  MoveL 10746 to (-26.41, 164.46, 144.49) mm, rotated rx 180 ry 0 rz 180 deg; joints [-138.58, 73.769, -86.473, 137.874, 80.508, 8.483]
  MoveL 10747 to (-26.41, 164.46, 144.49) mm, rotated rx 180 ry 0 rz 180 deg; joints [-138.58, 73.769, -86.473, 137.874, 80.508, 8.483]
  Call Extruder(786.45061)
  MoveL 10748 to (-26.72, 164.41, 144.49) mm, rotated rx 180 ry 0 rz 180 deg; joints [-138.635, 73.783, -86.46, 137.932, 80.52, 8.455]
  MoveL 10749 to (-26.72, 164.41, 144.49) mm, rotated rx 180 ry 0 rz 180 deg; joints [-138.635, 73.783, -86.46, 137.932, 80.52, 8.455]
  Call Extruder(786.61308)
  MoveL 10750 to (-27.03, 164.37, 144.49) mm, rotated rx -180 ry 0 rz -180 deg; joints [-138.69, 73.796, -86.447, 137.99, 80.531, 8.428]
  MoveL 10751 to (-27.03, 164.37, 144.49) mm, rotated rx -180 ry 0 rz -180 deg; joints [-138.69, 73.796, -86.447, 137.99, 80.531, 8.428]
  Call Extruder(786.74701)
  MoveL 10752 to (-27.27, 164.32, 144.49) mm, rotated rx -180 ry 0 rz 180 deg; joints [-138.736, 73.807, -86.437, 138.039, 80.54, 8.407]
  MoveL 10753 to (-27.27, 164.32, 144.49) mm, rotated rx -180 ry 0 rz 180 deg; joints [-138.736, 73.807, -86.437, 138.039, 80.54, 8.407]
  Call Extruder(786.88155)
  MoveL 10754 to (-27.52, 164.27, 144.49) mm, rotated rx -180 ry 0 rz 180 deg; joints [-138.783, 73.817, -86.426, 138.088, 80.549, 8.385]
  MoveL 10755 to (-27.52, 164.27, 144.49) mm, rotated rx -180 ry 0 rz 180 deg; joints [-138.783, 73.817, -86.426, 138.088, 80.549, 8.385]
  Call Extruder(787.01669)
  MoveL 10756 to (-27.77, 164.22, 144.49) mm, rotated rx 180 ry 0 rz -180 deg; joints [-138.829, 73.828, -86.416, 138.137, 80.557, 8.363]
  MoveL 10757 to (-27.77, 164.22, 144.49) mm, rotated rx 180 ry 0 rz -180 deg; joints [-138.829, 73.828, -86.416, 138.137, 80.557, 8.363]
  Call Extruder(787.15245)
  MoveL 10758 to (-28.02, 164.17, 144.49) mm, rotated rx -180 ry 0 rz 180 deg; joints [-138.875, 73.838, -86.406, 138.185, 80.566, 8.342]
  MoveL 10759 to (-28.02, 164.17, 144.49) mm, rotated rx -180 ry 0 rz 180 deg; joints [-138.875, 73.838, -86.406, 138.185, 80.566, 8.342]
  Call Extruder(787.28882)
  MoveL 10760 to (-28.27, 164.12, 144.49) mm, rotated rx -180 ry 0 rz 180 deg; joints [-138.921, 73.848, -86.395, 138.234, 80.575, 8.32]
  MoveL 10761 to (-28.27, 164.12, 144.49) mm, rotated rx -180 ry 0 rz 180 deg; joints [-138.921, 73.848, -86.395, 138.234, 80.575, 8.32]
  Call Extruder(787.42580)
  MoveL 10762 to (-28.52, 164.07, 144.49) mm, rotated rx -180 ry 0 rz 180 deg; joints [-138.967, 73.859, -86.385, 138.283, 80.584, 8.298]
  MoveL 10763 to (-28.52, 164.07, 144.49) mm, rotated rx -180 ry 0 rz 180 deg; joints [-138.967, 73.859, -86.385, 138.283, 80.584, 8.298]
  Call Extruder(787.56338)
  MoveL 10764 to (-28.77, 164.02, 144.49) mm, rotated rx -180 ry 0 rz 180 deg; joints [-139.013, 73.869, -86.375, 138.331, 80.593, 8.277]
  MoveL 10765 to (-28.77, 164.02, 144.49) mm, rotated rx -180 ry 0 rz 180 deg; joints [-139.013, 73.869, -86.375, 138.331, 80.593, 8.277]
  Call Extruder(787.67710)
  MoveL 10766 to (-28.97, 163.97, 144.49) mm, rotated rx -180 ry 0 rz -180 deg; joints [-139.052, 73.878, -86.366, 138.371, 80.6, 8.259]
  MoveL 10767 to (-28.97, 163.97, 144.49) mm, rotated rx -180 ry 0 rz -180 deg; joints [-139.052, 73.878, -86.366, 138.371, 80.6, 8.259]
  Call Extruder(787.79127)
  MoveL 10768 to (-29.18, 163.93, 144.49) mm, rotated rx -180 ry 0 rz 180 deg; joints [-139.09, 73.886, -86.358, 138.412, 80.607, 8.241]
  MoveL 10769 to (-29.18, 163.93, 144.49) mm, rotated rx -180 ry 0 rz 180 deg; joints [-139.09, 73.886, -86.358, 138.412, 80.607, 8.241]
  Call Extruder(787.90589)
  MoveL 10770 to (-29.38, 163.88, 144.49) mm, rotated rx 180 ry 0 rz 180 deg; joints [-139.128, 73.895, -86.349, 138.452, 80.614, 8.224]
  MoveL 10771 to (-29.38, 163.88, 144.49) mm, rotated rx 180 ry 0 rz 180 deg; joints [-139.128, 73.895, -86.349, 138.452, 80.614, 8.224]
  Call Extruder(788.02096)
  MoveL 10772 to (-29.59, 163.84, 144.49) mm, rotated rx 180 ry 0 rz 180 deg; joints [-139.166, 73.903, -86.341, 138.492, 80.621, 8.206]
  MoveL 10773 to (-29.59, 163.84, 144.49) mm, rotated rx 180 ry 0 rz 180 deg; joints [-139.166, 73.903, -86.341, 138.492, 80.621, 8.206]
  Call Extruder(788.14320)
  MoveL 10774 to (-29.8, 163.78, 144.49) mm, rotated rx -180 ry 0 rz -180 deg; joints [-139.208, 73.911, -86.332, 138.536, 80.628, 8.188]
  MoveL 10775 to (-29.8, 163.78, 144.49) mm, rotated rx -180 ry 0 rz -180 deg; joints [-139.208, 73.911, -86.332, 138.536, 80.628, 8.188]
  Call Extruder(788.27288)
  MoveL 10776 to (-30.02, 163.72, 144.49) mm, rotated rx -180 ry 0 rz 180 deg; joints [-139.253, 73.92, -86.324, 138.583, 80.634, 8.17]
  MoveL 10777 to (-30.02, 163.72, 144.49) mm, rotated rx -180 ry 0 rz 180 deg; joints [-139.253, 73.92, -86.324, 138.583, 80.634, 8.17]
  Call Extruder(788.40312)
  MoveL 10778 to (-30.25, 163.65, 144.49) mm, rotated rx -180 ry 0 rz 180 deg; joints [-139.298, 73.928, -86.316, 138.63, 80.64, 8.151]
  MoveL 10779 to (-30.25, 163.65, 144.49) mm, rotated rx -180 ry 0 rz 180 deg; joints [-139.298, 73.928, -86.316, 138.63, 80.64, 8.151]
  Call Extruder(788.53393)
  MoveL 10780 to (-30.47, 163.58, 144.49) mm, rotated rx -180 ry 0 rz 180 deg; joints [-139.343, 73.937, -86.307, 138.677, 80.647, 8.132]
  MoveL 10781 to (-30.47, 163.58, 144.49) mm, rotated rx -180 ry 0 rz 180 deg; joints [-139.343, 73.937, -86.307, 138.677, 80.647, 8.132]
  Call Extruder(788.66530)
  MoveL 10782 to (-30.69, 163.51, 144.49) mm, rotated rx -180 ry 0 rz 180 deg; joints [-139.388, 73.945, -86.299, 138.724, 80.653, 8.114]
  MoveL 10783 to (-30.69, 163.51, 144.49) mm, rotated rx -180 ry 0 rz 180 deg; joints [-139.388, 73.945, -86.299, 138.724, 80.653, 8.114]
  Call Extruder(788.77719)
  MoveL 10784 to (-30.88, 163.45, 144.49) mm, rotated rx -180 ry 0 rz 180 deg; joints [-139.427, 73.952, -86.292, 138.764, 80.658, 8.098]
  MoveL 10785 to (-30.88, 163.45, 144.49) mm, rotated rx -180 ry 0 rz 180 deg; joints [-139.427, 73.952, -86.292, 138.764, 80.658, 8.098]
  Call Extruder(788.88953)
  MoveL 10786 to (-31.07, 163.39, 144.49) mm, rotated rx -180 ry 0 rz 180 deg; joints [-139.465, 73.959, -86.285, 138.804, 80.663, 8.083]
  MoveL 10787 to (-31.07, 163.39, 144.49) mm, rotated rx -180 ry 0 rz 180 deg; joints [-139.465, 73.959, -86.285, 138.804, 80.663, 8.083]
  Call Extruder(789.00231)
  MoveL 10788 to (-31.26, 163.33, 144.49) mm, rotated rx 180 ry 0 rz -180 deg; joints [-139.504, 73.966, -86.278, 138.844, 80.668, 8.067]
  MoveL 10789 to (-31.26, 163.33, 144.49) mm, rotated rx 180 ry 0 rz -180 deg; joints [-139.504, 73.966, -86.278, 138.844, 80.668, 8.067]
  Call Extruder(789.11553)
  MoveL 10790 to (-31.45, 163.27, 144.49) mm, rotated rx 180 ry 0 rz -180 deg; joints [-139.542, 73.973, -86.271, 138.885, 80.673, 8.052]
  MoveL 10791 to (-31.45, 163.27, 144.49) mm, rotated rx 180 ry 0 rz -180 deg; joints [-139.542, 73.973, -86.271, 138.885, 80.673, 8.052]
  Call Extruder(789.22920)
  MoveL 10792 to (-31.64, 163.21, 144.49) mm, rotated rx 180 ry 0 rz 180 deg; joints [-139.581, 73.979, -86.264, 138.925, 80.678, 8.036]
  MoveL 10793 to (-31.64, 163.21, 144.49) mm, rotated rx 180 ry 0 rz 180 deg; joints [-139.581, 73.979, -86.264, 138.925, 80.678, 8.036]
  Call Extruder(789.41118)
  MoveL 10794 to (-31.93, 163.09, 144.49) mm, rotated rx -180 ry 0 rz -180 deg; joints [-139.645, 73.989, -86.254, 138.991, 80.684, 8.013]
  MoveL 10795 to (-31.93, 163.09, 144.49) mm, rotated rx -180 ry 0 rz -180 deg; joints [-139.645, 73.989, -86.254, 138.991, 80.684, 8.013]
  Call Extruder(789.59392)
  MoveL 10796 to (-32.22, 162.96, 144.49) mm, rotated rx -180 ry 0 rz 180 deg; joints [-139.709, 73.999, -86.244, 139.057, 80.69, 7.989]
  MoveL 10797 to (-32.22, 162.96, 144.49) mm, rotated rx -180 ry 0 rz 180 deg; joints [-139.709, 73.999, -86.244, 139.057, 80.69, 7.989]
  Call Extruder(789.76433)
  MoveL 10798 to (-32.49, 162.85, 144.49) mm, rotated rx 180 ry 0 rz -180 deg; joints [-139.768, 74.007, -86.235, 139.119, 80.695, 7.968]
  MoveL 10799 to (-32.49, 162.85, 144.49) mm, rotated rx 180 ry 0 rz -180 deg; joints [-139.768, 74.007, -86.235, 139.119, 80.695, 7.968]
  Call Extruder(789.92231)
  MoveL 10800 to (-32.74, 162.74, 144.49) mm, rotated rx 180 ry 0 rz 180 deg; joints [-139.823, 74.016, -86.227, 139.176, 80.699, 7.948]
  MoveL 10801 to (-32.74, 162.74, 144.49) mm, rotated rx 180 ry 0 rz 180 deg; joints [-139.823, 74.016, -86.227, 139.176, 80.699, 7.948]
  Call Extruder(790.08088)
  MoveL 10802 to (-32.99, 162.64, 144.49) mm, rotated rx -180 ry 0 rz -180 deg; joints [-139.878, 74.024, -86.219, 139.233, 80.704, 7.929]
  MoveL 10803 to (-32.99, 162.64, 144.49) mm, rotated rx -180 ry 0 rz -180 deg; joints [-139.878, 74.024, -86.219, 139.233, 80.704, 7.929]
  Call Extruder(790.28705)
  MoveL 10804 to (-33.29, 162.46, 144.49) mm, rotated rx 180 ry 0 rz 180 deg; joints [-139.953, 74.032, -86.211, 139.31, 80.706, 7.906]
  MoveL 10805 to (-33.29, 162.46, 144.49) mm, rotated rx 180 ry 0 rz 180 deg; joints [-139.953, 74.032, -86.211, 139.31, 80.706, 7.906]
  Call Extruder(790.49399)
  MoveL 10806 to (-33.6, 162.29, 144.49) mm, rotated rx -180 ry 0 rz -180 deg; joints [-140.028, 74.04, -86.202, 139.387, 80.708, 7.883]
  MoveL 10807 to (-33.6, 162.29, 144.49) mm, rotated rx -180 ry 0 rz -180 deg; joints [-140.028, 74.04, -86.202, 139.387, 80.708, 7.883]
  Call Extruder(790.70172)
  MoveL 10808 to (-33.9, 162.11, 144.49) mm, rotated rx 180 ry 0 rz 180 deg; joints [-140.103, 74.048, -86.194, 139.463, 80.71, 7.86]
  MoveL 10809 to (-33.9, 162.11, 144.49) mm, rotated rx 180 ry 0 rz 180 deg; joints [-140.103, 74.048, -86.194, 139.463, 80.71, 7.86]
  Call Extruder(790.91022)
  MoveL 10810 to (-34.21, 161.94, 144.49) mm, rotated rx 180 ry 0 rz 180 deg; joints [-140.178, 74.056, -86.186, 139.54, 80.712, 7.837]
  MoveL 10811 to (-34.21, 161.94, 144.49) mm, rotated rx 180 ry 0 rz 180 deg; joints [-140.178, 74.056, -86.186, 139.54, 80.712, 7.837]
  Call Extruder(791.08976)
  MoveL 10812 to (-34.45, 161.76, 144.49) mm, rotated rx 180 ry 0 rz 180 deg; joints [-140.244, 74.061, -86.181, 139.607, 80.711, 7.82]
  MoveL 10813 to (-34.45, 161.76, 144.49) mm, rotated rx 180 ry 0 rz 180 deg; joints [-140.244, 74.061, -86.181, 139.607, 80.711, 7.82]
  Call Extruder(791.42319)
  MoveL 10814 to (-34.9, 161.43, 144.49) mm, rotated rx -180 ry 0 rz -180 deg; joints [-140.366, 74.07, -86.171, 139.732, 80.708, 7.788]
  MoveL 10815 to (-34.9, 161.43, 144.49) mm, rotated rx -180 ry 0 rz -180 deg; joints [-140.366, 74.07, -86.171, 139.732, 80.708, 7.788]
  Call Extruder(791.75781)
  MoveL 10816 to (-35.35, 161.1, 144.49) mm, rotated rx 180 ry 0 rz 180 deg; joints [-140.489, 74.079, -86.162, 139.857, 80.706, 7.756]
  Call Extruder(792.58572)
  MoveL 10817 to (-36.39, 160.19, 144.49) mm, rotated rx -180 ry 0 rz -180 deg; joints [-140.797, 74.094, -86.147, 140.17, 80.688, 7.686]
  Call Extruder(793.10708)
  MoveL 10818 to (-36.97, 159.54, 144.49) mm, rotated rx 180 ry 0 rz -180 deg; joints [-140.993, 74.096, -86.144, 140.368, 80.665, 7.651]
  Set speed (130.0 mm/s)
  MoveL 10819 to (-38.97, 156.79, 144.49) mm, rotated rx 180 ry 0 rz 180 deg; joints [-141.763, 74.086, -86.155, 141.139, 80.548, 7.538]
  MoveL 10820 to (-38.97, 156.78, 153.89) mm, rotated rx -180 ry 0 rz 180 deg; joints [-141.763, 75.445, -87.86, 141.102, 80.278, 7.758]
  Call Extruder(791.10708)
  Set speed (40.0 mm/s)
  MoveL 10821 to (-38.97, 156.78, 153.89) mm, rotated rx -180 ry 0 rz 180 deg; joints [-141.763, 75.445, -87.86, 141.102, 80.278, 7.758]
  Call Extruder(0.00000)
  Set speed (130.0 mm/s)
  MoveL 10822 to (-31.64, 163.21, 153.89) mm, rotated rx 180 ry 0 rz -180 deg; joints [-139.581, 75.337, -87.97, 138.886, 80.415, 8.268]
  Call Extruder(2.00000)
  Set speed (40.0 mm/s)
  MoveL 10823 to (-31.64, 163.21, 153.89) mm, rotated rx 180 ry 0 rz -180 deg; joints [-139.581, 75.337, -87.97, 138.886, 80.415, 8.268]
  Set speed (30.0 mm/s)
  MoveL 10824 to (-31.64, 163.21, 153.89) mm, rotated rx 180 ry 0 rz -180 deg; joints [-139.581, 75.337, -87.97, 138.886, 80.415, 8.268]
  Call Extruder(2.18198)
  MoveL 10825 to (-31.93, 163.09, 153.89) mm, rotated rx -180 ry 0 rz -180 deg; joints [-139.645, 75.347, -87.96, 138.953, 80.421, 8.245]
  MoveL 10826 to (-31.93, 163.09, 153.89) mm, rotated rx -180 ry 0 rz -180 deg; joints [-139.645, 75.347, -87.96, 138.953, 80.421, 8.245]
  Call Extruder(2.36471)
  MoveL 10827 to (-32.22, 162.96, 153.89) mm, rotated rx -180 ry 0 rz -180 deg; joints [-139.709, 75.356, -87.95, 139.019, 80.427, 8.221]
  MoveL 10828 to (-32.22, 162.96, 153.89) mm, rotated rx -180 ry 0 rz -180 deg; joints [-139.709, 75.356, -87.95, 139.019, 80.427, 8.221]
  Call Extruder(2.53265)
  MoveL 10829 to (-32.49, 162.85, 153.89) mm, rotated rx 180 ry 0 rz 180 deg; joints [-139.767, 75.365, -87.941, 139.08, 80.432, 8.199]
  MoveL 10830 to (-32.49, 162.85, 153.89) mm, rotated rx 180 ry 0 rz 180 deg; joints [-139.767, 75.365, -87.941, 139.08, 80.432, 8.199]
  Call Extruder(2.68564)
  MoveL 10831 to (-32.73, 162.75, 153.89) mm, rotated rx -180 ry 0 rz 180 deg; joints [-139.821, 75.373, -87.933, 139.135, 80.436, 8.18]
  MoveL 10832 to (-32.73, 162.75, 153.89) mm, rotated rx -180 ry 0 rz 180 deg; joints [-139.821, 75.373, -87.933, 139.135, 80.436, 8.18]
  Call Extruder(2.83919)
  MoveL 10833 to (-32.97, 162.65, 153.89) mm, rotated rx 180 ry 0 rz 180 deg; joints [-139.874, 75.381, -87.925, 139.19, 80.441, 8.16]
  MoveL 10834 to (-32.97, 162.65, 153.89) mm, rotated rx 180 ry 0 rz 180 deg; joints [-139.874, 75.381, -87.925, 139.19, 80.441, 8.16]
  Call Extruder(3.04828)
  MoveL 10835 to (-33.28, 162.47, 153.89) mm, rotated rx -180 ry 0 rz 180 deg; joints [-139.95, 75.389, -87.917, 139.269, 80.442, 8.137]
  MoveL 10836 to (-33.28, 162.47, 153.89) mm, rotated rx -180 ry 0 rz 180 deg; joints [-139.95, 75.389, -87.917, 139.269, 80.442, 8.137]
  Call Extruder(3.25817)
  MoveL 10837 to (-33.59, 162.29, 153.89) mm, rotated rx -180 ry 0 rz -180 deg; joints [-140.026, 75.398, -87.909, 139.347, 80.444, 8.113]
  MoveL 10838 to (-33.59, 162.29, 153.89) mm, rotated rx -180 ry 0 rz -180 deg; joints [-140.026, 75.398, -87.909, 139.347, 80.444, 8.113]
  Call Extruder(3.46884)
  MoveL 10839 to (-33.89, 162.11, 153.89) mm, rotated rx -180 ry 0 rz -180 deg; joints [-140.102, 75.406, -87.9, 139.425, 80.446, 8.09]
  MoveL 10840 to (-33.89, 162.11, 153.89) mm, rotated rx -180 ry 0 rz -180 deg; joints [-140.102, 75.406, -87.9, 139.425, 80.446, 8.09]
  Call Extruder(3.68030)
  MoveL 10841 to (-34.2, 161.93, 153.89) mm, rotated rx -180 ry 0 rz 180 deg; joints [-140.178, 75.414, -87.892, 139.503, 80.448, 8.066]
  MoveL 10842 to (-34.2, 161.93, 153.89) mm, rotated rx -180 ry 0 rz 180 deg; joints [-140.178, 75.414, -87.892, 139.503, 80.448, 8.066]
  Call Extruder(3.88506)
  MoveL 10843 to (-34.48, 161.73, 153.89) mm, rotated rx -180 ry 0 rz -180 deg; joints [-140.253, 75.42, -87.886, 139.579, 80.447, 8.045]
  MoveL 10844 to (-34.48, 161.73, 153.89) mm, rotated rx -180 ry 0 rz -180 deg; joints [-140.253, 75.42, -87.886, 139.579, 80.447, 8.045]
  Call Extruder(4.20602)
  MoveL 10845 to (-34.92, 161.42, 153.89) mm, rotated rx 180 ry 0 rz 180 deg; joints [-140.371, 75.429, -87.877, 139.7, 80.444, 8.014]
  MoveL 10846 to (-34.92, 161.42, 153.89) mm, rotated rx 180 ry 0 rz 180 deg; joints [-140.371, 75.429, -87.877, 139.7, 80.444, 8.014]
  Call Extruder(4.52807)
  MoveL 10847 to (-35.35, 161.1, 153.89) mm, rotated rx 180 ry 0 rz 180 deg; joints [-140.489, 75.438, -87.867, 139.82, 80.442, 7.982]
  Call Extruder(5.35599)
  MoveL 10848 to (-36.39, 160.19, 153.89) mm, rotated rx -180 ry 0 rz 180 deg; joints [-140.797, 75.453, -87.852, 140.133, 80.422, 7.911]
  Call Extruder(6.18392)
  MoveL 10849 to (-37.3, 159.15, 153.89) mm, rotated rx 180 ry 0 rz 180 deg; joints [-141.109, 75.457, -87.848, 140.447, 80.385, 7.854]
  Call Extruder(6.34862)
  MoveL 10850 to (-37.47, 158.93, 153.89) mm, rotated rx -180 ry 0 rz -180 deg; joints [-141.171, 75.456, -87.849, 140.509, 80.375, 7.845]
  MoveL 10851 to (-37.47, 158.93, 153.89) mm, rotated rx -180 ry 0 rz -180 deg; joints [-141.171, 75.456, -87.849, 140.509, 80.375, 7.845]
  Call Extruder(6.67688)
  MoveL 10852 to (-37.79, 158.49, 153.89) mm, rotated rx -180 ry 0 rz 180 deg; joints [-141.295, 75.454, -87.851, 140.634, 80.356, 7.826]
  MoveL 10853 to (-37.79, 158.49, 153.89) mm, rotated rx -180 ry 0 rz 180 deg; joints [-141.295, 75.454, -87.851, 140.634, 80.356, 7.826]
  Call Extruder(7.00398)
  MoveL 10854 to (-38.11, 158.04, 153.89) mm, rotated rx -180 ry 0 rz -180 deg; joints [-141.419, 75.452, -87.853, 140.758, 80.336, 7.807]
  MoveL 10855 to (-38.11, 158.04, 153.89) mm, rotated rx -180 ry 0 rz -180 deg; joints [-141.419, 75.452, -87.853, 140.758, 80.336, 7.807]
  Call Extruder(7.13851)
  MoveL 10856 to (-38.23, 157.85, 153.89) mm, rotated rx 180 ry 0 rz 180 deg; joints [-141.47, 75.45, -87.855, 140.808, 80.326, 7.802]
  MoveL 10857 to (-38.23, 157.85, 153.89) mm, rotated rx 180 ry 0 rz 180 deg; joints [-141.47, 75.45, -87.855, 140.808, 80.326, 7.802]
  Call Extruder(7.35382)
  MoveL 10858 to (-38.41, 157.53, 153.89) mm, rotated rx -180 ry 0 rz 180 deg; joints [-141.551, 75.447, -87.859, 140.889, 80.309, 7.793]
  MoveL 10859 to (-38.41, 157.53, 153.89) mm, rotated rx -180 ry 0 rz 180 deg; joints [-141.551, 75.447, -87.859, 140.889, 80.309, 7.793]
  Call Extruder(7.56829)
  MoveL 10860 to (-38.59, 157.22, 153.89) mm, rotated rx -180 ry 0 rz -180 deg; joints [-141.632, 75.443, -87.863, 140.97, 80.292, 7.784]
  MoveL 10861 to (-38.59, 157.22, 153.89) mm, rotated rx -180 ry 0 rz -180 deg; joints [-141.632, 75.443, -87.863, 140.97, 80.292, 7.784]
  Call Extruder(7.78192)
  MoveL 10862 to (-38.77, 156.9, 153.89) mm, rotated rx -180 ry 0 rz 180 deg; joints [-141.714, 75.439, -87.866, 141.051, 80.275, 7.775]
  MoveL 10863 to (-38.77, 156.9, 153.89) mm, rotated rx -180 ry 0 rz 180 deg; joints [-141.714, 75.439, -87.866, 141.051, 80.275, 7.775]
  Call Extruder(7.96114)
  MoveL 10864 to (-38.91, 156.63, 153.89) mm, rotated rx -180 ry 0 rz 180 deg; joints [-141.782, 75.435, -87.87, 141.119, 80.26, 7.768]
  MoveL 10865 to (-38.91, 156.63, 153.89) mm, rotated rx -180 ry 0 rz 180 deg; joints [-141.782, 75.435, -87.87, 141.119, 80.26, 7.768]
  Call Extruder(8.10685)
  MoveL 10866 to (-39.01, 156.4, 153.89) mm, rotated rx -180 ry 0 rz -180 deg; joints [-141.837, 75.431, -87.875, 141.173, 80.246, 7.764]
  MoveL 10867 to (-39.01, 156.4, 153.89) mm, rotated rx -180 ry 0 rz -180 deg; joints [-141.837, 75.431, -87.875, 141.173, 80.246, 7.764]
  Call Extruder(8.25205)
  MoveL 10868 to (-39.11, 156.17, 153.89) mm, rotated rx 180 ry 0 rz 180 deg; joints [-141.891, 75.427, -87.879, 141.227, 80.232, 7.761]
  MoveL 10869 to (-39.11, 156.17, 153.89) mm, rotated rx 180 ry 0 rz 180 deg; joints [-141.891, 75.427, -87.879, 141.227, 80.232, 7.761]
  Call Extruder(8.43477)
  MoveL 10870 to (-39.23, 155.88, 153.89) mm, rotated rx 180 ry 0 rz -180 deg; joints [-141.96, 75.421, -87.885, 141.295, 80.213, 7.756]
  MoveL 10871 to (-39.23, 155.88, 153.89) mm, rotated rx 180 ry 0 rz -180 deg; joints [-141.96, 75.421, -87.885, 141.295, 80.213, 7.756]
  Call Extruder(8.61673)
  MoveL 10872 to (-39.35, 155.58, 153.89) mm, rotated rx -180 ry 0 rz 180 deg; joints [-142.029, 75.415, -87.891, 141.363, 80.195, 7.752]
  MoveL 10873 to (-39.35, 155.58, 153.89) mm, rotated rx -180 ry 0 rz 180 deg; joints [-142.029, 75.415, -87.891, 141.363, 80.195, 7.752]
  Call Extruder(8.76407)
  MoveL 10874 to (-39.44, 155.34, 153.89) mm, rotated rx -180 ry 0 rz 180 deg; joints [-142.085, 75.41, -87.896, 141.418, 80.179, 7.749]
  MoveL 10875 to (-39.44, 155.34, 153.89) mm, rotated rx -180 ry 0 rz 180 deg; joints [-142.085, 75.41, -87.896, 141.418, 80.179, 7.749]
  Call Extruder(8.87730)
  MoveL 10876 to (-39.5, 155.15, 153.89) mm, rotated rx -180 ry 0 rz -180 deg; joints [-142.127, 75.405, -87.901, 141.46, 80.166, 7.747]
  MoveL 10877 to (-39.5, 155.15, 153.89) mm, rotated rx -180 ry 0 rz -180 deg; joints [-142.127, 75.405, -87.901, 141.46, 80.166, 7.747]
  Call Extruder(8.99009)
  MoveL 10878 to (-39.56, 154.97, 153.89) mm, rotated rx -180 ry 0 rz -180 deg; joints [-142.169, 75.401, -87.905, 141.501, 80.154, 7.746]
  MoveL 10879 to (-39.56, 154.97, 153.89) mm, rotated rx -180 ry 0 rz -180 deg; joints [-142.169, 75.401, -87.905, 141.501, 80.154, 7.746]
  Call Extruder(9.10244)
  MoveL 10880 to (-39.62, 154.78, 153.89) mm, rotated rx 180 ry 0 rz -180 deg; joints [-142.212, 75.396, -87.91, 141.543, 80.141, 7.744]
  MoveL 10881 to (-39.62, 154.78, 153.89) mm, rotated rx 180 ry 0 rz -180 deg; joints [-142.212, 75.396, -87.91, 141.543, 80.141, 7.744]
  Call Extruder(9.21434)
  MoveL 10882 to (-39.68, 154.59, 153.89) mm, rotated rx 180 ry 0 rz -180 deg; joints [-142.254, 75.392, -87.914, 141.584, 80.128, 7.743]
  MoveL 10883 to (-39.68, 154.59, 153.89) mm, rotated rx 180 ry 0 rz -180 deg; joints [-142.254, 75.392, -87.914, 141.584, 80.128, 7.743]
  Call Extruder(9.33574)
  MoveL 10884 to (-39.75, 154.38, 153.89) mm, rotated rx -180 ry 0 rz 180 deg; joints [-142.3, 75.387, -87.919, 141.629, 80.114, 7.741]
  MoveL 10885 to (-39.75, 154.38, 153.89) mm, rotated rx -180 ry 0 rz 180 deg; joints [-142.3, 75.387, -87.919, 141.629, 80.114, 7.741]
  Call Extruder(9.46653)
  MoveL 10886 to (-39.81, 154.16, 153.89) mm, rotated rx -180 ry 0 rz 180 deg; joints [-142.35, 75.381, -87.925, 141.678, 80.098, 7.74]
  MoveL 10887 to (-39.81, 154.16, 153.89) mm, rotated rx -180 ry 0 rz 180 deg; joints [-142.35, 75.381, -87.925, 141.678, 80.098, 7.74]
  Call Extruder(9.59676)
  MoveL 10888 to (-39.88, 153.94, 153.89) mm, rotated rx -180 ry 0 rz -180 deg; joints [-142.399, 75.376, -87.931, 141.726, 80.083, 7.738]
  MoveL 10889 to (-39.88, 153.94, 153.89) mm, rotated rx -180 ry 0 rz -180 deg; joints [-142.399, 75.376, -87.931, 141.726, 80.083, 7.738]
  Call Extruder(9.72643)
  MoveL 10890 to (-39.95, 153.71, 153.89) mm, rotated rx -180 ry 0 rz 180 deg; joints [-142.449, 75.37, -87.936, 141.775, 80.067, 7.737]
  MoveL 10891 to (-39.95, 153.71, 153.89) mm, rotated rx -180 ry 0 rz 180 deg; joints [-142.449, 75.37, -87.936, 141.775, 80.067, 7.737]
  Call Extruder(9.85553)
  MoveL 10892 to (-40.02, 153.49, 153.89) mm, rotated rx -180 ry 0 rz -180 deg; joints [-142.498, 75.364, -87.942, 141.824, 80.052, 7.735]
  MoveL 10893 to (-40.02, 153.49, 153.89) mm, rotated rx -180 ry 0 rz -180 deg; joints [-142.498, 75.364, -87.942, 141.824, 80.052, 7.735]
  Call Extruder(9.97061)
  MoveL 10894 to (-40.06, 153.28, 153.89) mm, rotated rx 180 ry 0 rz -180 deg; joints [-142.541, 75.358, -87.948, 141.866, 80.036, 7.735]
  MoveL 10895 to (-40.06, 153.28, 153.89) mm, rotated rx 180 ry 0 rz -180 deg; joints [-142.541, 75.358, -87.948, 141.866, 80.036, 7.735]
  Call Extruder(10.08525)
  MoveL 10896 to (-40.11, 153.08, 153.89) mm, rotated rx -180 ry 0 rz 180 deg; joints [-142.584, 75.352, -87.954, 141.908, 80.021, 7.735]
  MoveL 10897 to (-40.11, 153.08, 153.89) mm, rotated rx -180 ry 0 rz 180 deg; joints [-142.584, 75.352, -87.954, 141.908, 80.021, 7.735]
  Call Extruder(10.19943)
  MoveL 10898 to (-40.15, 152.88, 153.89) mm, rotated rx -180 ry 0 rz 180 deg; joints [-142.627, 75.346, -87.96, 141.95, 80.006, 7.735]
  MoveL 10899 to (-40.15, 152.88, 153.89) mm, rotated rx -180 ry 0 rz 180 deg; joints [-142.627, 75.346, -87.96, 141.95, 80.006, 7.735]
  Call Extruder(10.31316)
  MoveL 10900 to (-40.2, 152.67, 153.89) mm, rotated rx -180 ry 0 rz -180 deg; joints [-142.671, 75.34, -87.966, 141.992, 79.991, 7.735]
  MoveL 10901 to (-40.2, 152.67, 153.89) mm, rotated rx -180 ry 0 rz -180 deg; joints [-142.671, 75.34, -87.966, 141.992, 79.991, 7.735]
  Call Extruder(10.43859)
  MoveL 10902 to (-40.24, 152.44, 153.89) mm, rotated rx -180 ry 0 rz 180 deg; joints [-142.718, 75.334, -87.973, 142.038, 79.974, 7.736]
  MoveL 10903 to (-40.24, 152.44, 153.89) mm, rotated rx -180 ry 0 rz 180 deg; joints [-142.718, 75.334, -87.973, 142.038, 79.974, 7.736]
  Call Extruder(10.57556)
  MoveL 10904 to (-40.29, 152.2, 153.89) mm, rotated rx 180 ry 0 rz -180 deg; joints [-142.77, 75.326, -87.981, 142.089, 79.955, 7.736]
  MoveL 10905 to (-40.29, 152.2, 153.89) mm, rotated rx 180 ry 0 rz -180 deg; joints [-142.77, 75.326, -87.981, 142.089, 79.955, 7.736]
  Call Extruder(10.71193)
  MoveL 10906 to (-40.34, 151.95, 153.89) mm, rotated rx -180 ry 0 rz 180 deg; joints [-142.822, 75.318, -87.988, 142.14, 79.936, 7.736]
  MoveL 10907 to (-40.34, 151.95, 153.89) mm, rotated rx -180 ry 0 rz 180 deg; joints [-142.822, 75.318, -87.988, 142.14, 79.936, 7.736]
  Call Extruder(10.84768)
  MoveL 10908 to (-40.39, 151.7, 153.89) mm, rotated rx 180 ry 0 rz 180 deg; joints [-142.874, 75.311, -87.996, 142.191, 79.917, 7.736]
  MoveL 10909 to (-40.39, 151.7, 153.89) mm, rotated rx 180 ry 0 rz 180 deg; joints [-142.874, 75.311, -87.996, 142.191, 79.917, 7.736]
  Call Extruder(10.98283)
  MoveL 10910 to (-40.44, 151.45, 153.89) mm, rotated rx 180 ry 0 rz 180 deg; joints [-142.926, 75.303, -88.003, 142.241, 79.898, 7.737]
  MoveL 10911 to (-40.44, 151.45, 153.89) mm, rotated rx 180 ry 0 rz 180 deg; joints [-142.926, 75.303, -88.003, 142.241, 79.898, 7.737]
  Call Extruder(11.11736)
  MoveL 10912 to (-40.49, 151.2, 153.89) mm, rotated rx -180 ry 0 rz 180 deg; joints [-142.978, 75.296, -88.011, 142.292, 79.879, 7.737]
  MoveL 10913 to (-40.49, 151.2, 153.89) mm, rotated rx -180 ry 0 rz 180 deg; joints [-142.978, 75.296, -88.011, 142.292, 79.879, 7.737]
  Call Extruder(11.25129)
  MoveL 10914 to (-40.54, 150.95, 153.89) mm, rotated rx -180 ry 0 rz -180 deg; joints [-143.031, 75.288, -88.018, 142.343, 79.86, 7.737]
  MoveL 10915 to (-40.54, 150.95, 153.89) mm, rotated rx -180 ry 0 rz -180 deg; joints [-143.031, 75.288, -88.018, 142.343, 79.86, 7.737]
  Call Extruder(11.39914)
  MoveL 10916 to (-40.59, 150.67, 153.89) mm, rotated rx -180 ry 0 rz 180 deg; joints [-143.088, 75.28, -88.027, 142.399, 79.839, 7.737]
  MoveL 10917 to (-40.59, 150.67, 153.89) mm, rotated rx -180 ry 0 rz 180 deg; joints [-143.088, 75.28, -88.027, 142.399, 79.839, 7.737]
  Call Extruder(11.56087)
  MoveL 10918 to (-40.64, 150.37, 153.89) mm, rotated rx -180 ry 0 rz 180 deg; joints [-143.15, 75.27, -88.037, 142.46, 79.815, 7.738]
  MoveL 10919 to (-40.64, 150.37, 153.89) mm, rotated rx -180 ry 0 rz 180 deg; joints [-143.15, 75.27, -88.037, 142.46, 79.815, 7.738]
  Call Extruder(11.72186)
  MoveL 10920 to (-40.69, 150.06, 153.89) mm, rotated rx -180 ry 0 rz -180 deg; joints [-143.213, 75.26, -88.046, 142.521, 79.791, 7.739]
  MoveL 10921 to (-40.69, 150.06, 153.89) mm, rotated rx -180 ry 0 rz -180 deg; joints [-143.213, 75.26, -88.046, 142.521, 79.791, 7.739]
  Call Extruder(11.88213)
  MoveL 10922 to (-40.74, 149.76, 153.89) mm, rotated rx 180 ry 0 rz 180 deg; joints [-143.276, 75.25, -88.056, 142.582, 79.767, 7.74]
  MoveL 10923 to (-40.74, 149.76, 153.89) mm, rotated rx 180 ry 0 rz 180 deg; joints [-143.276, 75.25, -88.056, 142.582, 79.767, 7.74]
  Call Extruder(12.04168)
  MoveL 10924 to (-40.78, 149.45, 153.89) mm, rotated rx 180 ry 0 rz 180 deg; joints [-143.338, 75.24, -88.066, 142.643, 79.743, 7.741]
  MoveL 10925 to (-40.78, 149.45, 153.89) mm, rotated rx 180 ry 0 rz 180 deg; joints [-143.338, 75.24, -88.066, 142.643, 79.743, 7.741]
  Call Extruder(12.20049)
  MoveL 10926 to (-40.83, 149.14, 153.89) mm, rotated rx -180 ry 0 rz -180 deg; joints [-143.401, 75.23, -88.075, 142.704, 79.719, 7.742]
  MoveL 10927 to (-40.83, 149.14, 153.89) mm, rotated rx -180 ry 0 rz -180 deg; joints [-143.401, 75.23, -88.075, 142.704, 79.719, 7.742]
  Call Extruder(12.37915)
  MoveL 10928 to (-40.88, 148.8, 153.89) mm, rotated rx 180 ry 0 rz -180 deg; joints [-143.471, 75.219, -88.087, 142.772, 79.691, 7.743]
  MoveL 10929 to (-40.88, 148.8, 153.89) mm, rotated rx 180 ry 0 rz -180 deg; joints [-143.471, 75.219, -88.087, 142.772, 79.691, 7.743]
  Call Extruder(12.57759)
  MoveL 10930 to (-40.92, 148.41, 153.89) mm, rotated rx -180 ry 0 rz 180 deg; joints [-143.549, 75.206, -88.1, 142.847, 79.66, 7.745]
  MoveL 10931 to (-40.92, 148.41, 153.89) mm, rotated rx -180 ry 0 rz 180 deg; joints [-143.549, 75.206, -88.1, 142.847, 79.66, 7.745]
  Call Extruder(12.77517)
  MoveL 10932 to (-40.97, 148.02, 153.89) mm, rotated rx -180 ry 0 rz -180 deg; joints [-143.627, 75.192, -88.113, 142.923, 79.628, 7.747]
  MoveL 10933 to (-40.97, 148.02, 153.89) mm, rotated rx -180 ry 0 rz -180 deg; joints [-143.627, 75.192, -88.113, 142.923, 79.628, 7.747]
  Call Extruder(12.97187)
  MoveL 10934 to (-41.02, 147.63, 153.89) mm, rotated rx -180 ry 0 rz -180 deg; joints [-143.705, 75.179, -88.126, 142.998, 79.597, 7.749]
  MoveL 10935 to (-41.02, 147.63, 153.89) mm, rotated rx -180 ry 0 rz -180 deg; joints [-143.705, 75.179, -88.126, 142.998, 79.597, 7.749]
  Call Extruder(13.16771)
  MoveL 10936 to (-41.06, 147.25, 153.89) mm, rotated rx 180 ry 0 rz 180 deg; joints [-143.783, 75.166, -88.139, 143.074, 79.565, 7.751]
  MoveL 10937 to (-41.06, 147.25, 153.89) mm, rotated rx 180 ry 0 rz 180 deg; joints [-143.783, 75.166, -88.139, 143.074, 79.565, 7.751]
  Call Extruder(13.46311)
  MoveL 10938 to (-41.11, 146.66, 153.89) mm, rotated rx 180 ry 0 rz 180 deg; joints [-143.899, 75.145, -88.159, 143.186, 79.516, 7.756]
  MoveL 10939 to (-41.11, 146.66, 153.89) mm, rotated rx 180 ry 0 rz 180 deg; joints [-143.899, 75.145, -88.159, 143.186, 79.516, 7.756]
  Call Extruder(13.75718)
  MoveL 10940 to (-41.15, 146.07, 153.89) mm, rotated rx -180 ry 0 rz 180 deg; joints [-144.015, 75.123, -88.18, 143.298, 79.467, 7.76]
  MoveL 10941 to (-41.15, 146.07, 153.89) mm, rotated rx -180 ry 0 rz 180 deg; joints [-144.015, 75.123, -88.18, 143.298, 79.467, 7.76]
  Call Extruder(14.04991)
  MoveL 10942 to (-41.2, 145.48, 153.89) mm, rotated rx 180 ry 0 rz 180 deg; joints [-144.131, 75.102, -88.201, 143.411, 79.417, 7.764]
  MoveL 10943 to (-41.2, 145.48, 153.89) mm, rotated rx 180 ry 0 rz 180 deg; joints [-144.131, 75.102, -88.201, 143.411, 79.417, 7.764]
  Call Extruder(14.62336)
  MoveL 10944 to (-41.25, 144.32, 153.89) mm, rotated rx -180 ry 0 rz -180 deg; joints [-144.355, 75.058, -88.243, 143.627, 79.317, 7.775]
  MoveL 10945 to (-41.25, 144.32, 153.89) mm, rotated rx -180 ry 0 rz -180 deg; joints [-144.355, 75.058, -88.243, 143.627, 79.317, 7.775]
  Call Extruder(15.33742)
  MoveL 10946 to (-41.29, 142.86, 153.89) mm, rotated rx -180 ry 0 rz -180 deg; joints [-144.635, 75.001, -88.297, 143.897, 79.19, 7.788]
  Call Extruder(57.40821)
  MoveL 10947 to (-41.29, 57.14, 153.89) mm, rotated rx 180 ry 0 rz 180 deg; joints [-164.153, 72.135, -90.522, 163.346, 72.335, 5.187]
  Call Extruder(57.85446)
  MoveL 10948 to (-41.27, 56.23, 153.89) mm, rotated rx 180 ry 0 rz 180 deg; joints [-164.391, 72.113, -90.536, 163.592, 72.279, 5.122]
  MoveL 10949 to (-41.27, 56.23, 153.89) mm, rotated rx 180 ry 0 rz 180 deg; joints [-164.391, 72.113, -90.536, 163.592, 72.279, 5.122]
  Call Extruder(58.44013)
  MoveL 10950 to (-41.22, 55.04, 153.89) mm, rotated rx 180 ry 0 rz 180 deg; joints [-164.701, 72.083, -90.555, 163.912, 72.205, 5.037]
  MoveL 10951 to (-41.22, 55.04, 153.89) mm, rotated rx 180 ry 0 rz 180 deg; joints [-164.701, 72.083, -90.555, 163.912, 72.205, 5.037]
  Call Extruder(58.87777)
  MoveL 10952 to (-41.17, 54.16, 153.89) mm, rotated rx -180 ry 0 rz -180 deg; joints [-164.932, 72.06, -90.569, 164.15, 72.149, 4.974]
  MoveL 10953 to (-41.17, 54.16, 153.89) mm, rotated rx -180 ry 0 rz -180 deg; joints [-164.932, 72.06, -90.569, 164.15, 72.149, 4.974]
  Call Extruder(59.16609)
  MoveL 10954 to (-41.13, 53.58, 153.89) mm, rotated rx 180 ry 0 rz -180 deg; joints [-165.082, 72.044, -90.579, 164.305, 72.11, 4.933]
  MoveL 10955 to (-41.13, 53.58, 153.89) mm, rotated rx 180 ry 0 rz -180 deg; joints [-165.082, 72.044, -90.579, 164.305, 72.11, 4.933]
  Call Extruder(59.45571)
  MoveL 10956 to (-41.08, 53, 153.89) mm, rotated rx -180 ry 0 rz 180 deg; joints [-165.233, 72.028, -90.589, 164.461, 72.073, 4.892]
  MoveL 10957 to (-41.08, 53, 153.89) mm, rotated rx -180 ry 0 rz 180 deg; joints [-165.233, 72.028, -90.589, 164.461, 72.073, 4.892]
  Call Extruder(59.69701)
  MoveL 10958 to (-41.04, 52.53, 153.89) mm, rotated rx -180 ry 0 rz -180 deg; joints [-165.357, 72.014, -90.598, 164.589, 72.041, 4.858]
  MoveL 10959 to (-41.04, 52.53, 153.89) mm, rotated rx -180 ry 0 rz -180 deg; joints [-165.357, 72.014, -90.598, 164.589, 72.041, 4.858]
  Call Extruder(59.88962)
  MoveL 10960 to (-40.99, 52.15, 153.89) mm, rotated rx -180 ry 0 rz 180 deg; joints [-165.455, 72.002, -90.605, 164.69, 72.014, 4.832]
  MoveL 10961 to (-40.99, 52.15, 153.89) mm, rotated rx -180 ry 0 rz 180 deg; joints [-165.455, 72.002, -90.605, 164.69, 72.014, 4.832]
  Call Extruder(60.08307)
  MoveL 10962 to (-40.95, 51.77, 153.89) mm, rotated rx -180 ry 0 rz -180 deg; joints [-165.554, 71.991, -90.612, 164.792, 71.988, 4.805]
  MoveL 10963 to (-40.95, 51.77, 153.89) mm, rotated rx -180 ry 0 rz -180 deg; joints [-165.554, 71.991, -90.612, 164.792, 71.988, 4.805]
  Call Extruder(60.27736)
  MoveL 10964 to (-40.9, 51.39, 153.89) mm, rotated rx -180 ry 0 rz -180 deg; joints [-165.652, 71.979, -90.619, 164.893, 71.962, 4.778]
  MoveL 10965 to (-40.9, 51.39, 153.89) mm, rotated rx -180 ry 0 rz -180 deg; joints [-165.652, 71.979, -90.619, 164.893, 71.962, 4.778]
  Call Extruder(60.47247)
  MoveL 10966 to (-40.86, 51.01, 153.89) mm, rotated rx 180 ry 0 rz -180 deg; joints [-165.751, 71.968, -90.626, 164.995, 71.936, 4.751]
  MoveL 10967 to (-40.86, 51.01, 153.89) mm, rotated rx 180 ry 0 rz -180 deg; joints [-165.751, 71.968, -90.626, 164.995, 71.936, 4.751]
  Call Extruder(60.63128)
  MoveL 10968 to (-40.81, 50.7, 153.89) mm, rotated rx -180 ry 0 rz -180 deg; joints [-165.829, 71.958, -90.633, 165.076, 71.913, 4.73]
  MoveL 10969 to (-40.81, 50.7, 153.89) mm, rotated rx -180 ry 0 rz -180 deg; joints [-165.829, 71.958, -90.633, 165.076, 71.913, 4.73]
  Call Extruder(60.79083)
  MoveL 10970 to (-40.76, 50.4, 153.89) mm, rotated rx 180 ry 0 rz 180 deg; joints [-165.908, 71.947, -90.639, 165.157, 71.891, 4.709]
  MoveL 10971 to (-40.76, 50.4, 153.89) mm, rotated rx 180 ry 0 rz 180 deg; joints [-165.908, 71.947, -90.639, 165.157, 71.891, 4.709]
  Call Extruder(60.95110)
  MoveL 10972 to (-40.71, 50.09, 153.89) mm, rotated rx -180 ry 0 rz -180 deg; joints [-165.987, 71.937, -90.645, 165.238, 71.869, 4.688]
  MoveL 10973 to (-40.71, 50.09, 153.89) mm, rotated rx -180 ry 0 rz -180 deg; joints [-165.987, 71.937, -90.645, 165.238, 71.869, 4.688]
  Call Extruder(61.11209)
  MoveL 10974 to (-40.66, 49.79, 153.89) mm, rotated rx 180 ry 0 rz 180 deg; joints [-166.066, 71.927, -90.651, 165.32, 71.846, 4.666]
  MoveL 10975 to (-40.66, 49.79, 153.89) mm, rotated rx 180 ry 0 rz 180 deg; joints [-166.066, 71.927, -90.651, 165.32, 71.846, 4.666]
  Call Extruder(61.27382)
  MoveL 10976 to (-40.61, 49.48, 153.89) mm, rotated rx 180 ry 0 rz 180 deg; joints [-166.145, 71.917, -90.657, 165.402, 71.824, 4.645]
  MoveL 10977 to (-40.61, 49.48, 153.89) mm, rotated rx 180 ry 0 rz 180 deg; joints [-166.145, 71.917, -90.657, 165.402, 71.824, 4.645]
  Call Extruder(61.43627)
  MoveL 10978 to (-40.57, 49.18, 153.89) mm, rotated rx 180 ry 0 rz -180 deg; joints [-166.224, 71.907, -90.664, 165.483, 71.802, 4.623]
  MoveL 10979 to (-40.57, 49.18, 153.89) mm, rotated rx 180 ry 0 rz -180 deg; joints [-166.224, 71.907, -90.664, 165.483, 71.802, 4.623]
  Call Extruder(61.57020)
  MoveL 10980 to (-40.52, 48.93, 153.89) mm, rotated rx -180 ry 0 rz -180 deg; joints [-166.288, 71.898, -90.669, 165.549, 71.783, 4.606]
  MoveL 10981 to (-40.52, 48.93, 153.89) mm, rotated rx -180 ry 0 rz -180 deg; joints [-166.288, 71.898, -90.669, 165.549, 71.783, 4.606]
  Call Extruder(61.70473)
  MoveL 10982 to (-40.47, 48.68, 153.89) mm, rotated rx 180 ry 0 rz 180 deg; joints [-166.352, 71.889, -90.674, 165.615, 71.764, 4.589]
  MoveL 10983 to (-40.47, 48.68, 153.89) mm, rotated rx 180 ry 0 rz 180 deg; joints [-166.352, 71.889, -90.674, 165.615, 71.764, 4.589]
  Call Extruder(61.83988)
  MoveL 10984 to (-40.42, 48.43, 153.89) mm, rotated rx -180 ry 0 rz -180 deg; joints [-166.416, 71.88, -90.68, 165.681, 71.745, 4.571]
  MoveL 10985 to (-40.42, 48.43, 153.89) mm, rotated rx -180 ry 0 rz -180 deg; joints [-166.416, 71.88, -90.68, 165.681, 71.745, 4.571]
  Call Extruder(61.97563)
  MoveL 10986 to (-40.37, 48.18, 153.89) mm, rotated rx 180 ry 0 rz 180 deg; joints [-166.48, 71.871, -90.685, 165.747, 71.726, 4.554]
  MoveL 10987 to (-40.37, 48.18, 153.89) mm, rotated rx 180 ry 0 rz 180 deg; joints [-166.48, 71.871, -90.685, 165.747, 71.726, 4.554]
  Call Extruder(62.11200)
  MoveL 10988 to (-40.32, 47.93, 153.89) mm, rotated rx 180 ry 0 rz 180 deg; joints [-166.544, 71.862, -90.691, 165.813, 71.707, 4.537]
  MoveL 10989 to (-40.32, 47.93, 153.89) mm, rotated rx 180 ry 0 rz 180 deg; joints [-166.544, 71.862, -90.691, 165.813, 71.707, 4.537]
  Call Extruder(62.24897)
  MoveL 10990 to (-40.27, 47.68, 153.89) mm, rotated rx -180 ry 0 rz -180 deg; joints [-166.608, 71.853, -90.696, 165.88, 71.688, 4.519]
  MoveL 10991 to (-40.27, 47.68, 153.89) mm, rotated rx -180 ry 0 rz -180 deg; joints [-166.608, 71.853, -90.696, 165.88, 71.688, 4.519]
  Call Extruder(62.38656)
  MoveL 10992 to (-40.22, 47.43, 153.89) mm, rotated rx -180 ry 0 rz -180 deg; joints [-166.673, 71.844, -90.702, 165.946, 71.669, 4.502]
  MoveL 10993 to (-40.22, 47.43, 153.89) mm, rotated rx -180 ry 0 rz -180 deg; joints [-166.673, 71.844, -90.702, 165.946, 71.669, 4.502]
  Call Extruder(62.50029)
  MoveL 10994 to (-40.17, 47.23, 153.89) mm, rotated rx 180 ry 0 rz -180 deg; joints [-166.725, 71.837, -90.706, 166, 71.653, 4.487]
  MoveL 10995 to (-40.17, 47.23, 153.89) mm, rotated rx 180 ry 0 rz -180 deg; joints [-166.725, 71.837, -90.706, 166, 71.653, 4.487]
  Call Extruder(62.61447)
  MoveL 10996 to (-40.13, 47.02, 153.89) mm, rotated rx -180 ry 0 rz 180 deg; joints [-166.778, 71.829, -90.711, 166.054, 71.637, 4.473]
  MoveL 10997 to (-40.13, 47.02, 153.89) mm, rotated rx -180 ry 0 rz 180 deg; joints [-166.778, 71.829, -90.711, 166.054, 71.637, 4.473]
  Call Extruder(62.72910)
  MoveL 10998 to (-40.08, 46.82, 153.89) mm, rotated rx 180 ry 0 rz 180 deg; joints [-166.83, 71.822, -90.715, 166.109, 71.621, 4.459]
  MoveL 10999 to (-40.08, 46.82, 153.89) mm, rotated rx 180 ry 0 rz 180 deg; joints [-166.83, 71.822, -90.715, 166.109, 71.621, 4.459]
  Call Extruder(62.84419)
  MoveL 11000 to (-40.04, 46.61, 153.89) mm, rotated rx -180 ry 0 rz -180 deg; joints [-166.883, 71.814, -90.72, 166.163, 71.606, 4.444]
  MoveL 11001 to (-40.04, 46.61, 153.89) mm, rotated rx -180 ry 0 rz -180 deg; joints [-166.883, 71.814, -90.72, 166.163, 71.606, 4.444]
  Call Extruder(62.96643)
  MoveL 11002 to (-39.98, 46.4, 153.89) mm, rotated rx -180 ry 0 rz -180 deg; joints [-166.937, 71.806, -90.725, 166.219, 71.588, 4.43]
  MoveL 11003 to (-39.98, 46.4, 153.89) mm, rotated rx -180 ry 0 rz -180 deg; joints [-166.937, 71.806, -90.725, 166.219, 71.588, 4.43]
  Call Extruder(63.09609)
  MoveL 11004 to (-39.92, 46.18, 153.89) mm, rotated rx -180 ry 0 rz -180 deg; joints [-166.994, 71.796, -90.731, 166.277, 71.568, 4.415]
  MoveL 11005 to (-39.92, 46.18, 153.89) mm, rotated rx -180 ry 0 rz -180 deg; joints [-166.994, 71.796, -90.731, 166.277, 71.568, 4.415]
  Call Extruder(63.22632)
  MoveL 11006 to (-39.85, 45.95, 153.89) mm, rotated rx -180 ry 0 rz 180 deg; joints [-167.051, 71.786, -90.737, 166.336, 71.549, 4.4]
  MoveL 11007 to (-39.85, 45.95, 153.89) mm, rotated rx -180 ry 0 rz 180 deg; joints [-167.051, 71.786, -90.737, 166.336, 71.549, 4.4]
  Call Extruder(63.35712)
  MoveL 11008 to (-39.78, 45.73, 153.89) mm, rotated rx 180 ry 0 rz 180 deg; joints [-167.107, 71.776, -90.743, 166.394, 71.529, 4.385]
  MoveL 11009 to (-39.78, 45.73, 153.89) mm, rotated rx 180 ry 0 rz 180 deg; joints [-167.107, 71.776, -90.743, 166.394, 71.529, 4.385]
  Call Extruder(63.48848)
  MoveL 11010 to (-39.71, 45.51, 153.89) mm, rotated rx 180 ry 0 rz 180 deg; joints [-167.164, 71.766, -90.749, 166.453, 71.51, 4.37]
  MoveL 11011 to (-39.71, 45.51, 153.89) mm, rotated rx 180 ry 0 rz 180 deg; joints [-167.164, 71.766, -90.749, 166.453, 71.51, 4.37]
  Call Extruder(63.60038)
  MoveL 11012 to (-39.65, 45.32, 153.89) mm, rotated rx -180 ry 0 rz -180 deg; joints [-167.212, 71.758, -90.754, 166.501, 71.493, 4.357]
  MoveL 11013 to (-39.65, 45.32, 153.89) mm, rotated rx -180 ry 0 rz -180 deg; joints [-167.212, 71.758, -90.754, 166.501, 71.493, 4.357]
  Call Extruder(63.71272)
  MoveL 11014 to (-39.59, 45.13, 153.89) mm, rotated rx -180 ry 0 rz -180 deg; joints [-167.26, 71.749, -90.759, 166.551, 71.476, 4.345]
  MoveL 11015 to (-39.59, 45.13, 153.89) mm, rotated rx -180 ry 0 rz -180 deg; joints [-167.26, 71.749, -90.759, 166.551, 71.476, 4.345]
  Call Extruder(63.82551)
  MoveL 11016 to (-39.53, 44.94, 153.89) mm, rotated rx 180 ry 0 rz 180 deg; joints [-167.307, 71.741, -90.764, 166.6, 71.459, 4.332]
  MoveL 11017 to (-39.53, 44.94, 153.89) mm, rotated rx 180 ry 0 rz 180 deg; joints [-167.307, 71.741, -90.764, 166.6, 71.459, 4.332]
  Call Extruder(63.93874)
  MoveL 11018 to (-39.47, 44.75, 153.89) mm, rotated rx 180 ry 0 rz -180 deg; joints [-167.355, 71.732, -90.769, 166.649, 71.442, 4.32]
  MoveL 11019 to (-39.47, 44.75, 153.89) mm, rotated rx 180 ry 0 rz -180 deg; joints [-167.355, 71.732, -90.769, 166.649, 71.442, 4.32]
  Call Extruder(64.05242)
  MoveL 11020 to (-39.41, 44.56, 153.89) mm, rotated rx -180 ry 0 rz -180 deg; joints [-167.403, 71.724, -90.774, 166.698, 71.425, 4.307]
  MoveL 11021 to (-39.41, 44.56, 153.89) mm, rotated rx -180 ry 0 rz -180 deg; joints [-167.403, 71.724, -90.774, 166.698, 71.425, 4.307]
  Call Extruder(64.23439)
  MoveL 11022 to (-39.29, 44.27, 153.89) mm, rotated rx -180 ry 0 rz -180 deg; joints [-167.475, 71.708, -90.783, 166.773, 71.396, 4.288]
  MoveL 11023 to (-39.29, 44.27, 153.89) mm, rotated rx -180 ry 0 rz -180 deg; joints [-167.475, 71.708, -90.783, 166.773, 71.396, 4.288]
  Call Extruder(64.41711)
  MoveL 11024 to (-39.17, 43.98, 153.89) mm, rotated rx 180 ry 0 rz 180 deg; joints [-167.548, 71.693, -90.792, 166.847, 71.367, 4.27]
  MoveL 11025 to (-39.17, 43.98, 153.89) mm, rotated rx 180 ry 0 rz 180 deg; joints [-167.548, 71.693, -90.792, 166.847, 71.367, 4.27]
  Call Extruder(64.58752)
  MoveL 11026 to (-39.05, 43.71, 153.89) mm, rotated rx 180 ry 0 rz -180 deg; joints [-167.615, 71.679, -90.801, 166.916, 71.34, 4.253]
  MoveL 11027 to (-39.05, 43.71, 153.89) mm, rotated rx 180 ry 0 rz -180 deg; joints [-167.615, 71.679, -90.801, 166.916, 71.34, 4.253]
  Call Extruder(64.74550)
  MoveL 11028 to (-38.94, 43.46, 153.89) mm, rotated rx -180 ry 0 rz 180 deg; joints [-167.677, 71.665, -90.809, 166.98, 71.314, 4.237]
  MoveL 11029 to (-38.94, 43.46, 153.89) mm, rotated rx -180 ry 0 rz 180 deg; joints [-167.677, 71.665, -90.809, 166.98, 71.314, 4.237]
  Call Extruder(64.90409)
  MoveL 11030 to (-38.84, 43.21, 153.89) mm, rotated rx 180 ry 0 rz 180 deg; joints [-167.739, 71.652, -90.817, 167.044, 71.289, 4.221]
  MoveL 11031 to (-38.84, 43.21, 153.89) mm, rotated rx 180 ry 0 rz 180 deg; joints [-167.739, 71.652, -90.817, 167.044, 71.289, 4.221]
  Call Extruder(65.11025)
  MoveL 11032 to (-38.66, 42.91, 153.89) mm, rotated rx -180 ry 0 rz -180 deg; joints [-167.813, 71.632, -90.828, 167.119, 71.253, 4.204]
  MoveL 11033 to (-38.66, 42.91, 153.89) mm, rotated rx -180 ry 0 rz -180 deg; joints [-167.813, 71.632, -90.828, 167.119, 71.253, 4.204]
  Call Extruder(65.31720)
  MoveL 11034 to (-38.49, 42.6, 153.89) mm, rotated rx -180 ry 0 rz 180 deg; joints [-167.886, 71.612, -90.84, 167.193, 71.216, 4.186]
  MoveL 11035 to (-38.49, 42.6, 153.89) mm, rotated rx -180 ry 0 rz 180 deg; joints [-167.886, 71.612, -90.84, 167.193, 71.216, 4.186]
  Call Extruder(65.52492)
  MoveL 11036 to (-38.31, 42.3, 153.89) mm, rotated rx 180 ry 0 rz -180 deg; joints [-167.96, 71.592, -90.852, 167.269, 71.18, 4.169]
  MoveL 11037 to (-38.31, 42.3, 153.89) mm, rotated rx 180 ry 0 rz -180 deg; joints [-167.96, 71.592, -90.852, 167.269, 71.18, 4.169]
  Call Extruder(65.73342)
  MoveL 11038 to (-38.14, 41.99, 153.89) mm, rotated rx -180 ry 0 rz -180 deg; joints [-168.033, 71.572, -90.863, 167.344, 71.144, 4.151]
  MoveL 11039 to (-38.14, 41.99, 153.89) mm, rotated rx -180 ry 0 rz -180 deg; joints [-168.033, 71.572, -90.863, 167.344, 71.144, 4.151]
  Call Extruder(65.91297)
  MoveL 11040 to (-37.96, 41.75, 153.89) mm, rotated rx -180 ry 0 rz -180 deg; joints [-168.091, 71.553, -90.874, 167.402, 71.11, 4.138]
  MoveL 11041 to (-37.96, 41.75, 153.89) mm, rotated rx -180 ry 0 rz -180 deg; joints [-168.091, 71.553, -90.874, 167.402, 71.11, 4.138]
  Call Extruder(66.24641)
  MoveL 11042 to (-37.63, 41.3, 153.89) mm, rotated rx -180 ry 0 rz 180 deg; joints [-168.197, 71.518, -90.895, 167.51, 71.048, 4.115]
  MoveL 11043 to (-37.63, 41.3, 153.89) mm, rotated rx -180 ry 0 rz 180 deg; joints [-168.197, 71.518, -90.895, 167.51, 71.048, 4.115]
  Call Extruder(66.58104)
  MoveL 11044 to (-37.3, 40.85, 153.89) mm, rotated rx 180 ry 0 rz 180 deg; joints [-168.304, 71.483, -90.915, 167.618, 70.986, 4.091]
  Call Extruder(67.40900)
  MoveL 11045 to (-36.39, 39.81, 153.89) mm, rotated rx -180 ry 0 rz 180 deg; joints [-168.541, 71.388, -90.969, 167.858, 70.825, 4.042]
  Call Extruder(68.06491)
  MoveL 11046 to (-35.57, 39.08, 153.89) mm, rotated rx -180 ry 0 rz -180 deg; joints [-168.699, 71.307, -91.015, 168.015, 70.689, 4.015]
  Call Extruder(68.40395)
  MoveL 11047 to (-35.13, 38.73, 153.89) mm, rotated rx 180 ry 0 rz 180 deg; joints [-168.773, 71.263, -91.04, 168.089, 70.618, 4.004]
  MoveL 11048 to (-35.13, 38.73, 153.89) mm, rotated rx 180 ry 0 rz 180 deg; joints [-168.773, 71.263, -91.04, 168.089, 70.618, 4.004]
  Call Extruder(68.73731)
  MoveL 11049 to (-34.68, 38.41, 153.89) mm, rotated rx -180 ry 0 rz -180 deg; joints [-168.84, 71.22, -91.064, 168.155, 70.546, 3.996]
  MoveL 11050 to (-34.68, 38.41, 153.89) mm, rotated rx -180 ry 0 rz -180 deg; joints [-168.84, 71.22, -91.064, 168.155, 70.546, 3.996]
  Call Extruder(69.06951)
  MoveL 11051 to (-34.22, 38.08, 153.89) mm, rotated rx 180 ry 0 rz -180 deg; joints [-168.907, 71.176, -91.088, 168.221, 70.475, 3.987]
  MoveL 11052 to (-34.22, 38.08, 153.89) mm, rotated rx 180 ry 0 rz -180 deg; joints [-168.907, 71.176, -91.088, 168.221, 70.475, 3.987]
  Call Extruder(69.24304)
  MoveL 11053 to (-33.97, 37.93, 153.89) mm, rotated rx 180 ry 0 rz 180 deg; joints [-168.935, 71.152, -91.101, 168.248, 70.437, 3.985]
  MoveL 11054 to (-33.97, 37.93, 153.89) mm, rotated rx 180 ry 0 rz 180 deg; joints [-168.935, 71.152, -91.101, 168.248, 70.437, 3.985]
  Call Extruder(69.46654)
  MoveL 11055 to (-33.64, 37.74, 153.89) mm, rotated rx 180 ry 0 rz 180 deg; joints [-168.971, 71.121, -91.119, 168.282, 70.387, 3.983]
  MoveL 11056 to (-33.64, 37.74, 153.89) mm, rotated rx 180 ry 0 rz 180 deg; joints [-168.971, 71.121, -91.119, 168.282, 70.387, 3.983]
  Call Extruder(69.68914)
  MoveL 11057 to (-33.32, 37.55, 153.89) mm, rotated rx 180 ry 0 rz 180 deg; joints [-169.007, 71.09, -91.135, 168.317, 70.337, 3.98]
  MoveL 11058 to (-33.32, 37.55, 153.89) mm, rotated rx 180 ry 0 rz 180 deg; joints [-169.007, 71.09, -91.135, 168.317, 70.337, 3.98]
  Call Extruder(69.91084)
  MoveL 11059 to (-32.99, 37.36, 153.89) mm, rotated rx 180 ry 0 rz -180 deg; joints [-169.043, 71.059, -91.152, 168.351, 70.288, 3.978]
  MoveL 11060 to (-32.99, 37.36, 153.89) mm, rotated rx 180 ry 0 rz -180 deg; joints [-169.043, 71.059, -91.152, 168.351, 70.288, 3.978]
  Call Extruder(70.07784)
  MoveL 11061 to (-32.73, 37.25, 153.89) mm, rotated rx -180 ry 0 rz 180 deg; joints [-169.061, 71.034, -91.166, 168.368, 70.25, 3.979]
  MoveL 11062 to (-32.73, 37.25, 153.89) mm, rotated rx -180 ry 0 rz 180 deg; joints [-169.061, 71.034, -91.166, 168.368, 70.25, 3.979]
  Call Extruder(70.24417)
  MoveL 11063 to (-32.46, 37.14, 153.89) mm, rotated rx -180 ry 0 rz 180 deg; joints [-169.078, 71.01, -91.179, 168.384, 70.212, 3.981]
  MoveL 11064 to (-32.46, 37.14, 153.89) mm, rotated rx -180 ry 0 rz 180 deg; joints [-169.078, 71.01, -91.179, 168.384, 70.212, 3.981]
  Call Extruder(70.41418)
  MoveL 11065 to (-32.19, 37.02, 153.89) mm, rotated rx 180 ry 0 rz 180 deg; joints [-169.096, 70.985, -91.192, 168.4, 70.173, 3.983]
  MoveL 11066 to (-32.19, 37.02, 153.89) mm, rotated rx 180 ry 0 rz 180 deg; joints [-169.096, 70.985, -91.192, 168.4, 70.173, 3.983]
  Call Extruder(70.58788)
  MoveL 11067 to (-31.92, 36.91, 153.89) mm, rotated rx -180 ry 0 rz 180 deg; joints [-169.114, 70.959, -91.206, 168.416, 70.133, 3.985]
  MoveL 11068 to (-31.92, 36.91, 153.89) mm, rotated rx -180 ry 0 rz 180 deg; joints [-169.114, 70.959, -91.206, 168.416, 70.133, 3.985]
  Call Extruder(70.76089)
  MoveL 11069 to (-31.64, 36.79, 153.89) mm, rotated rx 180 ry 0 rz 180 deg; joints [-169.132, 70.933, -91.22, 168.432, 70.093, 3.987]
  MoveL 11070 to (-31.64, 36.79, 153.89) mm, rotated rx 180 ry 0 rz 180 deg; joints [-169.132, 70.933, -91.22, 168.432, 70.093, 3.987]
  Call Extruder(70.87435)
  MoveL 11071 to (-31.45, 36.73, 153.89) mm, rotated rx -180 ry 0 rz 180 deg; joints [-169.139, 70.916, -91.229, 168.438, 70.066, 3.99]
  MoveL 11072 to (-31.45, 36.73, 153.89) mm, rotated rx -180 ry 0 rz 180 deg; joints [-169.139, 70.916, -91.229, 168.438, 70.066, 3.99]
  Call Extruder(70.98736)
  MoveL 11073 to (-31.26, 36.67, 153.89) mm, rotated rx -180 ry 0 rz 180 deg; joints [-169.146, 70.899, -91.238, 168.443, 70.04, 3.993]
  MoveL 11074 to (-31.26, 36.67, 153.89) mm, rotated rx -180 ry 0 rz 180 deg; joints [-169.146, 70.899, -91.238, 168.443, 70.04, 3.993]
  Call Extruder(71.09993)
  MoveL 11075 to (-31.07, 36.61, 153.89) mm, rotated rx 180 ry 0 rz -180 deg; joints [-169.154, 70.882, -91.248, 168.449, 70.013, 3.996]
  MoveL 11076 to (-31.07, 36.61, 153.89) mm, rotated rx 180 ry 0 rz -180 deg; joints [-169.154, 70.882, -91.248, 168.449, 70.013, 3.996]
  Call Extruder(71.21206)
  MoveL 11077 to (-30.88, 36.55, 153.89) mm, rotated rx -180 ry 0 rz -180 deg; joints [-169.161, 70.864, -91.257, 168.455, 69.987, 3.999]
  MoveL 11078 to (-30.88, 36.55, 153.89) mm, rotated rx -180 ry 0 rz -180 deg; joints [-169.161, 70.864, -91.257, 168.455, 69.987, 3.999]
  Call Extruder(71.32374)
  MoveL 11079 to (-30.7, 36.49, 153.89) mm, rotated rx 180 ry 0 rz 180 deg; joints [-169.168, 70.847, -91.266, 168.461, 69.961, 4.002]
  MoveL 11080 to (-30.7, 36.49, 153.89) mm, rotated rx 180 ry 0 rz 180 deg; joints [-169.168, 70.847, -91.266, 168.461, 69.961, 4.002]
  Call Extruder(71.45479)
  MoveL 11081 to (-30.47, 36.42, 153.89) mm, rotated rx 180 ry 0 rz 180 deg; joints [-169.175, 70.827, -91.277, 168.466, 69.93, 4.006]
  MoveL 11082 to (-30.47, 36.42, 153.89) mm, rotated rx 180 ry 0 rz 180 deg; joints [-169.175, 70.827, -91.277, 168.466, 69.93, 4.006]
  Call Extruder(71.58528)
  MoveL 11083 to (-30.25, 36.35, 153.89) mm, rotated rx -180 ry 0 rz 180 deg; joints [-169.182, 70.806, -91.287, 168.471, 69.899, 4.01]
  MoveL 11084 to (-30.25, 36.35, 153.89) mm, rotated rx -180 ry 0 rz 180 deg; joints [-169.182, 70.806, -91.287, 168.471, 69.899, 4.01]
  Call Extruder(71.71521)
  MoveL 11085 to (-30.02, 36.28, 153.89) mm, rotated rx 180 ry 0 rz -180 deg; joints [-169.19, 70.786, -91.298, 168.477, 69.867, 4.014]
  MoveL 11086 to (-30.02, 36.28, 153.89) mm, rotated rx 180 ry 0 rz -180 deg; joints [-169.19, 70.786, -91.298, 168.477, 69.867, 4.014]
  Call Extruder(71.84457)
  MoveL 11087 to (-29.8, 36.22, 153.89) mm, rotated rx -180 ry 0 rz -180 deg; joints [-169.197, 70.765, -91.309, 168.483, 69.836, 4.018]
  MoveL 11088 to (-29.8, 36.22, 153.89) mm, rotated rx -180 ry 0 rz -180 deg; joints [-169.197, 70.765, -91.309, 168.483, 69.836, 4.018]
  Call Extruder(71.96654)
  MoveL 11089 to (-29.59, 36.16, 153.89) mm, rotated rx 180 ry 0 rz 180 deg; joints [-169.202, 70.746, -91.319, 168.485, 69.807, 4.023]
  MoveL 11090 to (-29.59, 36.16, 153.89) mm, rotated rx 180 ry 0 rz 180 deg; joints [-169.202, 70.746, -91.319, 168.485, 69.807, 4.023]
  Call Extruder(72.08140)
  MoveL 11091 to (-29.38, 36.12, 153.89) mm, rotated rx -180 ry 0 rz 180 deg; joints [-169.203, 70.727, -91.329, 168.485, 69.779, 4.028]
  MoveL 11092 to (-29.38, 36.12, 153.89) mm, rotated rx -180 ry 0 rz 180 deg; joints [-169.203, 70.727, -91.329, 168.485, 69.779, 4.028]
  Call Extruder(72.19582)
  MoveL 11093 to (-29.18, 36.07, 153.89) mm, rotated rx 180 ry 0 rz 180 deg; joints [-169.205, 70.709, -91.338, 168.484, 69.752, 4.033]
  MoveL 11094 to (-29.18, 36.07, 153.89) mm, rotated rx 180 ry 0 rz 180 deg; joints [-169.205, 70.709, -91.338, 168.484, 69.752, 4.033]
  Call Extruder(72.30978)
  MoveL 11095 to (-28.97, 36.03, 153.89) mm, rotated rx 180 ry 0 rz -180 deg; joints [-169.207, 70.69, -91.348, 168.484, 69.724, 4.039]
  MoveL 11096 to (-28.97, 36.03, 153.89) mm, rotated rx 180 ry 0 rz -180 deg; joints [-169.207, 70.69, -91.348, 168.484, 69.724, 4.039]
  Call Extruder(72.42328)
  MoveL 11097 to (-28.77, 35.98, 153.89) mm, rotated rx 180 ry 0 rz 180 deg; joints [-169.208, 70.672, -91.357, 168.484, 69.697, 4.044]
  MoveL 11098 to (-28.77, 35.98, 153.89) mm, rotated rx 180 ry 0 rz 180 deg; joints [-169.208, 70.672, -91.357, 168.484, 69.697, 4.044]
  Call Extruder(72.56057)
  MoveL 11099 to (-28.52, 35.93, 153.89) mm, rotated rx -180 ry 0 rz -180 deg; joints [-169.209, 70.649, -91.369, 168.482, 69.663, 4.051]
  MoveL 11100 to (-28.52, 35.93, 153.89) mm, rotated rx -180 ry 0 rz -180 deg; joints [-169.209, 70.649, -91.369, 168.482, 69.663, 4.051]
  Call Extruder(72.69724)
  MoveL 11101 to (-28.27, 35.88, 153.89) mm, rotated rx 180 ry 0 rz -180 deg; joints [-169.209, 70.627, -91.38, 168.48, 69.63, 4.058]
  MoveL 11102 to (-28.27, 35.88, 153.89) mm, rotated rx 180 ry 0 rz -180 deg; joints [-169.209, 70.627, -91.38, 168.48, 69.63, 4.058]
  Call Extruder(72.83330)
  MoveL 11103 to (-28.02, 35.83, 153.89) mm, rotated rx -180 ry 0 rz 180 deg; joints [-169.21, 70.604, -91.392, 168.478, 69.596, 4.065]
  MoveL 11104 to (-28.02, 35.83, 153.89) mm, rotated rx -180 ry 0 rz 180 deg; joints [-169.21, 70.604, -91.392, 168.478, 69.596, 4.065]
  Call Extruder(72.96875)
  MoveL 11105 to (-27.77, 35.78, 153.89) mm, rotated rx 180 ry 0 rz -180 deg; joints [-169.21, 70.582, -91.403, 168.476, 69.563, 4.072]
  MoveL 11106 to (-27.77, 35.78, 153.89) mm, rotated rx 180 ry 0 rz -180 deg; joints [-169.21, 70.582, -91.403, 168.476, 69.563, 4.072]
  Call Extruder(73.10359)
  MoveL 11107 to (-27.52, 35.73, 153.89) mm, rotated rx -180 ry 0 rz 180 deg; joints [-169.211, 70.559, -91.415, 168.474, 69.529, 4.079]
  MoveL 11108 to (-27.52, 35.73, 153.89) mm, rotated rx -180 ry 0 rz 180 deg; joints [-169.211, 70.559, -91.415, 168.474, 69.529, 4.079]
  Call Extruder(73.23783)
  MoveL 11109 to (-27.28, 35.68, 153.89) mm, rotated rx 180 ry 0 rz -180 deg; joints [-169.212, 70.536, -91.426, 168.473, 69.496, 4.086]
  MoveL 11110 to (-27.28, 35.68, 153.89) mm, rotated rx 180 ry 0 rz -180 deg; joints [-169.212, 70.536, -91.426, 168.473, 69.496, 4.086]
  Call Extruder(73.37145)
  MoveL 11111 to (-27.03, 35.64, 153.89) mm, rotated rx -180 ry 0 rz -180 deg; joints [-169.212, 70.514, -91.438, 168.471, 69.462, 4.093]
  MoveL 11112 to (-27.03, 35.64, 153.89) mm, rotated rx -180 ry 0 rz -180 deg; joints [-169.212, 70.514, -91.438, 168.471, 69.462, 4.093]
  Call Extruder(73.53354)
  MoveL 11113 to (-26.72, 35.59, 153.89) mm, rotated rx 180 ry 0 rz 180 deg; joints [-169.21, 70.486, -91.452, 168.465, 69.422, 4.103]
  MoveL 11114 to (-26.72, 35.59, 153.89) mm, rotated rx 180 ry 0 rz 180 deg; joints [-169.21, 70.486, -91.452, 168.465, 69.422, 4.103]
  Call Extruder(73.69491)
  MoveL 11115 to (-26.41, 35.54, 153.89) mm, rotated rx -180 ry 0 rz 180 deg; joints [-169.207, 70.458, -91.466, 168.458, 69.382, 4.113]
  MoveL 11116 to (-26.41, 35.54, 153.89) mm, rotated rx -180 ry 0 rz 180 deg; joints [-169.207, 70.458, -91.466, 168.458, 69.382, 4.113]
  Call Extruder(73.85555)
  MoveL 11117 to (-26.11, 35.49, 153.89) mm, rotated rx 180 ry 0 rz 180 deg; joints [-169.204, 70.431, -91.48, 168.452, 69.341, 4.123]
  MoveL 11118 to (-26.11, 35.49, 153.89) mm, rotated rx 180 ry 0 rz 180 deg; joints [-169.204, 70.431, -91.48, 168.452, 69.341, 4.123]
  Call Extruder(74.01546)
  MoveL 11119 to (-25.8, 35.44, 153.89) mm, rotated rx -180 ry 0 rz 180 deg; joints [-169.201, 70.403, -91.493, 168.446, 69.301, 4.133]
  MoveL 11120 to (-25.8, 35.44, 153.89) mm, rotated rx -180 ry 0 rz 180 deg; joints [-169.201, 70.403, -91.493, 168.446, 69.301, 4.133]
  Call Extruder(74.17465)
  MoveL 11121 to (-25.5, 35.39, 153.89) mm, rotated rx -180 ry 0 rz -180 deg; joints [-169.198, 70.375, -91.507, 168.44, 69.26, 4.143]
  MoveL 11122 to (-25.5, 35.39, 153.89) mm, rotated rx -180 ry 0 rz -180 deg; joints [-169.198, 70.375, -91.507, 168.44, 69.26, 4.143]
  Call Extruder(74.33311)
  MoveL 11123 to (-25.19, 35.34, 153.89) mm, rotated rx -180 ry 0 rz -180 deg; joints [-169.195, 70.348, -91.521, 168.433, 69.22, 4.153]
  MoveL 11124 to (-25.19, 35.34, 153.89) mm, rotated rx -180 ry 0 rz -180 deg; joints [-169.195, 70.348, -91.521, 168.433, 69.22, 4.153]
  Call Extruder(74.53198)
  MoveL 11125 to (-24.8, 35.3, 153.89) mm, rotated rx -180 ry 0 rz 180 deg; joints [-169.187, 70.313, -91.538, 168.42, 69.169, 4.167]
  MoveL 11126 to (-24.8, 35.3, 153.89) mm, rotated rx -180 ry 0 rz 180 deg; joints [-169.187, 70.313, -91.538, 168.42, 69.169, 4.167]
  Call Extruder(74.72999)
  MoveL 11127 to (-24.42, 35.25, 153.89) mm, rotated rx 180 ry 0 rz -180 deg; joints [-169.178, 70.278, -91.555, 168.407, 69.119, 4.182]
  MoveL 11128 to (-24.42, 35.25, 153.89) mm, rotated rx 180 ry 0 rz -180 deg; joints [-169.178, 70.278, -91.555, 168.407, 69.119, 4.182]
  Call Extruder(74.92713)
  MoveL 11129 to (-24.03, 35.21, 153.89) mm, rotated rx 180 ry 0 rz -180 deg; joints [-169.17, 70.243, -91.572, 168.394, 69.068, 4.196]
  MoveL 11130 to (-24.03, 35.21, 153.89) mm, rotated rx 180 ry 0 rz -180 deg; joints [-169.17, 70.243, -91.572, 168.394, 69.068, 4.196]
  Call Extruder(75.12340)
  MoveL 11131 to (-23.64, 35.16, 153.89) mm, rotated rx 180 ry 0 rz -180 deg; joints [-169.161, 70.207, -91.589, 168.381, 69.018, 4.211]
  MoveL 11132 to (-23.64, 35.16, 153.89) mm, rotated rx 180 ry 0 rz -180 deg; joints [-169.161, 70.207, -91.589, 168.381, 69.018, 4.211]
  Call Extruder(75.36909)
  MoveL 11133 to (-23.15, 35.11, 153.89) mm, rotated rx -180 ry 0 rz 180 deg; joints [-169.147, 70.163, -91.611, 168.361, 68.955, 4.23]
  MoveL 11134 to (-23.15, 35.11, 153.89) mm, rotated rx -180 ry 0 rz 180 deg; joints [-169.147, 70.163, -91.611, 168.361, 68.955, 4.23]
  Call Extruder(75.66381)
  MoveL 11135 to (-22.56, 35.07, 153.89) mm, rotated rx -180 ry 0 rz 180 deg; joints [-169.127, 70.11, -91.636, 168.333, 68.879, 4.255]
  MoveL 11136 to (-22.56, 35.07, 153.89) mm, rotated rx -180 ry 0 rz 180 deg; joints [-169.127, 70.11, -91.636, 168.333, 68.879, 4.255]
  Call Extruder(75.95720)
  MoveL 11137 to (-21.97, 35.02, 153.89) mm, rotated rx 180 ry 0 rz 180 deg; joints [-169.107, 70.057, -91.661, 168.305, 68.804, 4.28]
  MoveL 11138 to (-21.97, 35.02, 153.89) mm, rotated rx 180 ry 0 rz 180 deg; joints [-169.107, 70.057, -91.661, 168.305, 68.804, 4.28]
  Call Extruder(76.39052)
  MoveL 11139 to (-21.1, 34.97, 153.89) mm, rotated rx -180 ry 0 rz -180 deg; joints [-169.069, 69.978, -91.699, 168.256, 68.693, 4.32]
  MoveL 11140 to (-21.1, 34.97, 153.89) mm, rotated rx -180 ry 0 rz -180 deg; joints [-169.069, 69.978, -91.699, 168.256, 68.693, 4.32]
  Call Extruder(76.96268)
  MoveL 11141 to (-19.94, 34.93, 153.89) mm, rotated rx -180 ry 0 rz -180 deg; joints [-169.014, 69.873, -91.747, 168.185, 68.546, 4.375]
  MoveL 11142 to (-19.94, 34.93, 153.89) mm, rotated rx -180 ry 0 rz -180 deg; joints [-169.014, 69.873, -91.747, 168.185, 68.546, 4.375]
  Call Extruder(77.39112)
  MoveL 11143 to (-19.06, 34.91, 153.89) mm, rotated rx -180 ry 0 rz -180 deg; joints [-168.967, 69.794, -91.784, 168.125, 68.437, 4.419]
  Call Extruder(194.20579)
  MoveL 11144 to (219.06, 34.91, 153.89) mm, rotated rx -180 ry 0 rz 160 deg; joints [-52.528, 62.66, -93.765, 74.917, 98.923, 29.921]
  Call Extruder(194.63413)
  MoveL 11145 to (219.94, 34.93, 153.89) mm, rotated rx 180 ry 0 rz 160 deg; joints [-52.184, 62.722, -93.757, 74.604, 99.076, 29.806]
  MoveL 11146 to (219.94, 34.93, 153.89) mm, rotated rx 180 ry 0 rz 160 deg; joints [-52.184, 62.722, -93.757, 74.604, 99.076, 29.806]
  Call Extruder(195.20742)
  MoveL 11147 to (221.1, 34.98, 153.89) mm, rotated rx -180 ry 0 rz 160 deg; joints [-51.737, 62.807, -93.746, 74.196, 99.272, 29.649]
  MoveL 11148 to (221.1, 34.98, 153.89) mm, rotated rx -180 ry 0 rz 160 deg; joints [-51.737, 62.807, -93.746, 74.196, 99.272, 29.649]
  Call Extruder(195.64158)
  MoveL 11149 to (221.97, 35.02, 153.89) mm, rotated rx 180 ry 0 rz 160 deg; joints [-51.408, 62.872, -93.736, 73.894, 99.414, 29.53]
  MoveL 11150 to (221.97, 35.02, 153.89) mm, rotated rx 180 ry 0 rz 160 deg; joints [-51.408, 62.872, -93.736, 73.894, 99.414, 29.53]
  Call Extruder(195.93548)
  MoveL 11151 to (222.56, 35.07, 153.89) mm, rotated rx -180 ry 0 rz 160 deg; joints [-51.194, 62.918, -93.73, 73.697, 99.505, 29.448]
  MoveL 11152 to (222.56, 35.07, 153.89) mm, rotated rx -180 ry 0 rz 160 deg; joints [-51.194, 62.918, -93.73, 73.697, 99.505, 29.448]
  Call Extruder(196.23072)
  MoveL 11153 to (223.15, 35.12, 153.89) mm, rotated rx 180 ry 0 rz 160 deg; joints [-50.981, 62.963, -93.724, 73.5, 99.595, 29.366]
  MoveL 11154 to (223.15, 35.12, 153.89) mm, rotated rx 180 ry 0 rz 160 deg; joints [-50.981, 62.963, -93.724, 73.5, 99.595, 29.366]
  Call Extruder(196.47684)
  MoveL 11155 to (223.64, 35.16, 153.89) mm, rotated rx -180 ry 0 rz 160 deg; joints [-50.807, 63.002, -93.718, 73.34, 99.667, 29.298]
  MoveL 11156 to (223.64, 35.16, 153.89) mm, rotated rx -180 ry 0 rz 160 deg; joints [-50.807, 63.002, -93.718, 73.34, 99.667, 29.298]
  Call Extruder(196.67350)
  MoveL 11157 to (224.03, 35.21, 153.89) mm, rotated rx 180 ry 0 rz 160 deg; joints [-50.674, 63.033, -93.714, 73.216, 99.722, 29.243]
  MoveL 11158 to (224.03, 35.21, 153.89) mm, rotated rx 180 ry 0 rz 160 deg; joints [-50.674, 63.033, -93.714, 73.216, 99.722, 29.243]
  Call Extruder(196.87102)
  MoveL 11159 to (224.42, 35.26, 153.89) mm, rotated rx 180 ry 0 rz 160 deg; joints [-50.541, 63.065, -93.709, 73.092, 99.776, 29.188]
  MoveL 11160 to (224.42, 35.26, 153.89) mm, rotated rx 180 ry 0 rz 160 deg; joints [-50.541, 63.065, -93.709, 73.092, 99.776, 29.188]
  Call Extruder(197.06941)
  MoveL 11161 to (224.8, 35.3, 153.89) mm, rotated rx -180 ry 0 rz 160 deg; joints [-50.408, 63.096, -93.704, 72.969, 99.83, 29.133]
  MoveL 11162 to (224.8, 35.3, 153.89) mm, rotated rx -180 ry 0 rz 160 deg; joints [-50.408, 63.096, -93.704, 72.969, 99.83, 29.133]
  Call Extruder(197.26866)
  MoveL 11163 to (225.19, 35.35, 153.89) mm, rotated rx 180 ry 0 rz 160 deg; joints [-50.276, 63.128, -93.7, 72.846, 99.884, 29.078]
  MoveL 11164 to (225.19, 35.35, 153.89) mm, rotated rx 180 ry 0 rz 160 deg; joints [-50.276, 63.128, -93.7, 72.846, 99.884, 29.078]
  Call Extruder(197.42740)
  MoveL 11165 to (225.5, 35.39, 153.89) mm, rotated rx -180 ry 0 rz 160 deg; joints [-50.177, 63.154, -93.696, 72.752, 99.923, 29.034]
  MoveL 11166 to (225.5, 35.39, 153.89) mm, rotated rx -180 ry 0 rz 160 deg; joints [-50.177, 63.154, -93.696, 72.752, 99.923, 29.034]
  Call Extruder(197.58687)
  MoveL 11167 to (225.8, 35.44, 153.89) mm, rotated rx 180 ry 0 rz 160 deg; joints [-50.078, 63.18, -93.692, 72.659, 99.963, 28.989]
  MoveL 11168 to (225.8, 35.44, 153.89) mm, rotated rx 180 ry 0 rz 160 deg; joints [-50.078, 63.18, -93.692, 72.659, 99.963, 28.989]
  Call Extruder(197.74706)
  MoveL 11169 to (226.11, 35.49, 153.89) mm, rotated rx 180 ry 0 rz 160 deg; joints [-49.979, 63.206, -93.688, 72.566, 100.001, 28.945]
  MoveL 11170 to (226.11, 35.49, 153.89) mm, rotated rx 180 ry 0 rz 160 deg; joints [-49.979, 63.206, -93.688, 72.566, 100.001, 28.945]
  Call Extruder(197.90798)
  MoveL 11171 to (226.41, 35.54, 153.89) mm, rotated rx 180 ry 0 rz 160 deg; joints [-49.88, 63.232, -93.684, 72.474, 100.04, 28.901]
  MoveL 11172 to (226.41, 35.54, 153.89) mm, rotated rx 180 ry 0 rz 160 deg; joints [-49.88, 63.232, -93.684, 72.474, 100.04, 28.901]
  Call Extruder(198.06962)
  MoveL 11173 to (226.72, 35.59, 153.89) mm, rotated rx 180 ry 0 rz 160 deg; joints [-49.782, 63.258, -93.68, 72.381, 100.078, 28.856]
  MoveL 11174 to (226.72, 35.59, 153.89) mm, rotated rx 180 ry 0 rz 160 deg; joints [-49.782, 63.258, -93.68, 72.381, 100.078, 28.856]
  Call Extruder(198.23200)
  MoveL 11175 to (227.02, 35.64, 153.89) mm, rotated rx -180 ry 0 rz 160 deg; joints [-49.685, 63.284, -93.676, 72.29, 100.116, 28.812]
  MoveL 11176 to (227.02, 35.64, 153.89) mm, rotated rx -180 ry 0 rz 160 deg; joints [-49.685, 63.284, -93.676, 72.29, 100.116, 28.812]
  Call Extruder(198.36589)
  MoveL 11177 to (227.27, 35.69, 153.89) mm, rotated rx 180 ry 0 rz 160 deg; joints [-49.608, 63.306, -93.673, 72.217, 100.145, 28.775]
  MoveL 11178 to (227.27, 35.69, 153.89) mm, rotated rx 180 ry 0 rz 160 deg; joints [-49.608, 63.306, -93.673, 72.217, 100.145, 28.775]
  Call Extruder(198.50039)
  MoveL 11179 to (227.52, 35.74, 153.89) mm, rotated rx 180 ry 0 rz 160 deg; joints [-49.532, 63.328, -93.669, 72.145, 100.174, 28.738]
  MoveL 11180 to (227.52, 35.74, 153.89) mm, rotated rx 180 ry 0 rz 160 deg; joints [-49.532, 63.328, -93.669, 72.145, 100.174, 28.738]
  Call Extruder(198.63550)
  MoveL 11181 to (227.77, 35.79, 153.89) mm, rotated rx 180 ry 0 rz 160 deg; joints [-49.456, 63.35, -93.666, 72.073, 100.203, 28.702]
  MoveL 11182 to (227.77, 35.79, 153.89) mm, rotated rx 180 ry 0 rz 160 deg; joints [-49.456, 63.35, -93.666, 72.073, 100.203, 28.702]
  Call Extruder(198.77122)
  MoveL 11183 to (228.02, 35.84, 153.89) mm, rotated rx -180 ry 0 rz 160 deg; joints [-49.381, 63.373, -93.662, 72.002, 100.231, 28.665]
  MoveL 11184 to (228.02, 35.84, 153.89) mm, rotated rx -180 ry 0 rz 160 deg; joints [-49.381, 63.373, -93.662, 72.002, 100.231, 28.665]
  Call Extruder(198.90755)
  MoveL 11185 to (228.27, 35.89, 153.89) mm, rotated rx -180 ry 0 rz 160 deg; joints [-49.306, 63.395, -93.659, 71.93, 100.259, 28.628]
  MoveL 11186 to (228.27, 35.89, 153.89) mm, rotated rx -180 ry 0 rz 160 deg; joints [-49.306, 63.395, -93.659, 71.93, 100.259, 28.628]
  Call Extruder(199.04449)
  MoveL 11187 to (228.52, 35.94, 153.89) mm, rotated rx 180 ry 0 rz 160 deg; joints [-49.231, 63.417, -93.655, 71.859, 100.287, 28.592]
  MoveL 11188 to (228.52, 35.94, 153.89) mm, rotated rx 180 ry 0 rz 160 deg; joints [-49.231, 63.417, -93.655, 71.859, 100.287, 28.592]
  Call Extruder(199.18204)
  MoveL 11189 to (228.77, 35.98, 153.89) mm, rotated rx 180 ry 0 rz 160 deg; joints [-49.156, 63.439, -93.652, 71.788, 100.314, 28.555]
  MoveL 11190 to (228.77, 35.98, 153.89) mm, rotated rx 180 ry 0 rz 160 deg; joints [-49.156, 63.439, -93.652, 71.788, 100.314, 28.555]
  Call Extruder(199.30492)
  MoveL 11191 to (228.99, 36.03, 153.89) mm, rotated rx -180 ry 0 rz 160 deg; joints [-49.092, 63.459, -93.648, 71.726, 100.338, 28.522]
  MoveL 11192 to (228.99, 36.03, 153.89) mm, rotated rx -180 ry 0 rz 160 deg; joints [-49.092, 63.459, -93.648, 71.726, 100.338, 28.522]
  Call Extruder(199.42833)
  MoveL 11193 to (229.21, 36.08, 153.89) mm, rotated rx -180 ry 0 rz 160 deg; joints [-49.028, 63.479, -93.645, 71.665, 100.361, 28.489]
  MoveL 11194 to (229.21, 36.08, 153.89) mm, rotated rx -180 ry 0 rz 160 deg; joints [-49.028, 63.479, -93.645, 71.665, 100.361, 28.489]
  Call Extruder(199.55228)
  MoveL 11195 to (229.43, 36.13, 153.89) mm, rotated rx -180 ry 0 rz 160 deg; joints [-48.963, 63.5, -93.642, 71.603, 100.385, 28.456]
  MoveL 11196 to (229.43, 36.13, 153.89) mm, rotated rx -180 ry 0 rz 160 deg; joints [-48.963, 63.5, -93.642, 71.603, 100.385, 28.456]
  Call Extruder(199.67675)
  MoveL 11197 to (229.65, 36.18, 153.89) mm, rotated rx 180 ry 0 rz 160 deg; joints [-48.9, 63.52, -93.639, 71.542, 100.408, 28.423]
  MoveL 11198 to (229.65, 36.18, 153.89) mm, rotated rx 180 ry 0 rz 160 deg; joints [-48.9, 63.52, -93.639, 71.542, 100.408, 28.423]
  Call Extruder(199.79915)
  MoveL 11199 to (229.87, 36.24, 153.89) mm, rotated rx -180 ry 0 rz 160 deg; joints [-48.841, 63.54, -93.635, 71.485, 100.428, 28.391]
  MoveL 11200 to (229.87, 36.24, 153.89) mm, rotated rx -180 ry 0 rz 160 deg; joints [-48.841, 63.54, -93.635, 71.485, 100.428, 28.391]
  Call Extruder(199.91963)
  MoveL 11201 to (230.07, 36.3, 153.89) mm, rotated rx 180 ry 0 rz 160 deg; joints [-48.786, 63.56, -93.632, 71.433, 100.446, 28.36]
  MoveL 11202 to (230.07, 36.3, 153.89) mm, rotated rx 180 ry 0 rz 160 deg; joints [-48.786, 63.56, -93.632, 71.433, 100.446, 28.36]
  Call Extruder(200.04059)
  MoveL 11203 to (230.28, 36.36, 153.89) mm, rotated rx 180 ry 0 rz 160 deg; joints [-48.732, 63.581, -93.629, 71.38, 100.465, 28.328]
  MoveL 11204 to (230.28, 36.36, 153.89) mm, rotated rx 180 ry 0 rz 160 deg; joints [-48.732, 63.581, -93.629, 71.38, 100.465, 28.328]
  Call Extruder(200.16205)
  MoveL 11205 to (230.49, 36.42, 153.89) mm, rotated rx 180 ry 0 rz 160 deg; joints [-48.678, 63.601, -93.625, 71.328, 100.483, 28.296]
  MoveL 11206 to (230.49, 36.42, 153.89) mm, rotated rx 180 ry 0 rz 160 deg; joints [-48.678, 63.601, -93.625, 71.328, 100.483, 28.296]
  Call Extruder(200.28400)
  MoveL 11207 to (230.7, 36.49, 153.89) mm, rotated rx 180 ry 0 rz 160 deg; joints [-48.624, 63.621, -93.622, 71.275, 100.501, 28.265]
  MoveL 11208 to (230.7, 36.49, 153.89) mm, rotated rx 180 ry 0 rz 160 deg; joints [-48.624, 63.621, -93.622, 71.275, 100.501, 28.265]
  Call Extruder(200.39590)
  MoveL 11209 to (230.88, 36.55, 153.89) mm, rotated rx -180 ry 0 rz 160 deg; joints [-48.577, 63.64, -93.619, 71.229, 100.516, 28.236]
  MoveL 11210 to (230.88, 36.55, 153.89) mm, rotated rx -180 ry 0 rz 160 deg; joints [-48.577, 63.64, -93.619, 71.229, 100.516, 28.236]
  Call Extruder(200.50825)
  MoveL 11211 to (231.07, 36.61, 153.89) mm, rotated rx 180 ry 0 rz 160 deg; joints [-48.529, 63.659, -93.616, 71.182, 100.531, 28.207]
  MoveL 11212 to (231.07, 36.61, 153.89) mm, rotated rx 180 ry 0 rz 160 deg; joints [-48.529, 63.659, -93.616, 71.182, 100.531, 28.207]
  Call Extruder(200.62104)
  MoveL 11213 to (231.26, 36.67, 153.89) mm, rotated rx -180 ry 0 rz 160 deg; joints [-48.482, 63.678, -93.613, 71.136, 100.546, 28.178]
  MoveL 11214 to (231.26, 36.67, 153.89) mm, rotated rx -180 ry 0 rz 160 deg; joints [-48.482, 63.678, -93.613, 71.136, 100.546, 28.178]
  Call Extruder(200.73427)
  MoveL 11215 to (231.45, 36.73, 153.89) mm, rotated rx -180 ry 0 rz 160 deg; joints [-48.435, 63.697, -93.609, 71.09, 100.562, 28.149]
  MoveL 11216 to (231.45, 36.73, 153.89) mm, rotated rx -180 ry 0 rz 160 deg; joints [-48.435, 63.697, -93.609, 71.09, 100.562, 28.149]
  Call Extruder(200.84795)
  MoveL 11217 to (231.64, 36.79, 153.89) mm, rotated rx 180 ry 0 rz 160 deg; joints [-48.388, 63.716, -93.606, 71.044, 100.577, 28.12]
  MoveL 11218 to (231.64, 36.79, 153.89) mm, rotated rx 180 ry 0 rz 160 deg; joints [-48.388, 63.716, -93.606, 71.044, 100.577, 28.12]
  Call Extruder(201.02990)
  MoveL 11219 to (231.93, 36.91, 153.89) mm, rotated rx 180 ry 0 rz 160 deg; joints [-48.324, 63.747, -93.601, 70.98, 100.595, 28.074]
  MoveL 11220 to (231.93, 36.91, 153.89) mm, rotated rx 180 ry 0 rz 160 deg; joints [-48.324, 63.747, -93.601, 70.98, 100.595, 28.074]
  Call Extruder(201.21262)
  MoveL 11221 to (232.22, 37.04, 153.89) mm, rotated rx 180 ry 0 rz 160 deg; joints [-48.259, 63.778, -93.596, 70.916, 100.613, 28.028]
  MoveL 11222 to (232.22, 37.04, 153.89) mm, rotated rx 180 ry 0 rz 160 deg; joints [-48.259, 63.778, -93.596, 70.916, 100.613, 28.028]
  Call Extruder(201.38304)
  MoveL 11223 to (232.49, 37.15, 153.89) mm, rotated rx 180 ry 0 rz 160 deg; joints [-48.201, 63.807, -93.591, 70.857, 100.629, 27.986]
  MoveL 11224 to (232.49, 37.15, 153.89) mm, rotated rx 180 ry 0 rz 160 deg; joints [-48.201, 63.807, -93.591, 70.857, 100.629, 27.986]
  Call Extruder(201.54104)
  MoveL 11225 to (232.74, 37.26, 153.89) mm, rotated rx 180 ry 0 rz 160 deg; joints [-48.148, 63.834, -93.586, 70.804, 100.644, 27.946]
  MoveL 11226 to (232.74, 37.26, 153.89) mm, rotated rx 180 ry 0 rz 160 deg; joints [-48.148, 63.834, -93.586, 70.804, 100.644, 27.946]
  Call Extruder(201.69964)
  MoveL 11227 to (232.99, 37.36, 153.89) mm, rotated rx 180 ry 0 rz 160 deg; joints [-48.095, 63.862, -93.581, 70.75, 100.658, 27.907]
  MoveL 11228 to (232.99, 37.36, 153.89) mm, rotated rx 180 ry 0 rz 160 deg; joints [-48.095, 63.862, -93.581, 70.75, 100.658, 27.907]
  Call Extruder(201.90581)
  MoveL 11229 to (233.29, 37.54, 153.89) mm, rotated rx 180 ry 0 rz 160 deg; joints [-48.044, 63.898, -93.575, 70.697, 100.668, 27.857]
  MoveL 11230 to (233.29, 37.54, 153.89) mm, rotated rx 180 ry 0 rz 160 deg; joints [-48.044, 63.898, -93.575, 70.697, 100.668, 27.857]
  Call Extruder(202.11275)
  MoveL 11231 to (233.6, 37.71, 153.89) mm, rotated rx 180 ry 0 rz 160 deg; joints [-47.994, 63.935, -93.568, 70.645, 100.677, 27.807]
  MoveL 11232 to (233.6, 37.71, 153.89) mm, rotated rx 180 ry 0 rz 160 deg; joints [-47.994, 63.935, -93.568, 70.645, 100.677, 27.807]
  Call Extruder(202.32048)
  MoveL 11233 to (233.9, 37.89, 153.89) mm, rotated rx -180 ry 0 rz 160 deg; joints [-47.944, 63.971, -93.562, 70.592, 100.686, 27.758]
  MoveL 11234 to (233.9, 37.89, 153.89) mm, rotated rx -180 ry 0 rz 160 deg; joints [-47.944, 63.971, -93.562, 70.592, 100.686, 27.758]
  Call Extruder(202.52898)
  MoveL 11235 to (234.21, 38.07, 153.89) mm, rotated rx 180 ry 0 rz 160 deg; joints [-47.895, 64.008, -93.555, 70.54, 100.694, 27.708]
  MoveL 11236 to (234.21, 38.07, 153.89) mm, rotated rx 180 ry 0 rz 160 deg; joints [-47.895, 64.008, -93.555, 70.54, 100.694, 27.708]
  Call Extruder(202.70852)
  MoveL 11237 to (234.45, 38.24, 153.89) mm, rotated rx 180 ry 0 rz 160 deg; joints [-47.866, 64.04, -93.549, 70.507, 100.695, 27.667]
  MoveL 11238 to (234.45, 38.24, 153.89) mm, rotated rx 180 ry 0 rz 160 deg; joints [-47.866, 64.04, -93.549, 70.507, 100.695, 27.667]
  Call Extruder(203.04194)
  MoveL 11239 to (234.9, 38.57, 153.89) mm, rotated rx -180 ry 0 rz 160 deg; joints [-47.814, 64.1, -93.538, 70.447, 100.696, 27.59]
  MoveL 11240 to (234.9, 38.57, 153.89) mm, rotated rx -180 ry 0 rz 160 deg; joints [-47.814, 64.1, -93.538, 70.447, 100.696, 27.59]
  Call Extruder(203.37654)
  MoveL 11241 to (235.35, 38.9, 153.89) mm, rotated rx -180 ry 0 rz 160 deg; joints [-47.762, 64.16, -93.527, 70.388, 100.696, 27.514]
  Call Extruder(204.20449)
  MoveL 11242 to (236.39, 39.81, 153.89) mm, rotated rx 180 ry 0 rz 160 deg; joints [-47.693, 64.309, -93.499, 70.294, 100.668, 27.332]
  Call Extruder(205.03243)
  MoveL 11243 to (237.3, 40.85, 153.89) mm, rotated rx 180 ry 0 rz -180 deg; joints [-27.851, 59.695, -94.019, 32.611, 119.904, 17.691]
  Call Extruder(205.19712)
  MoveL 11244 to (237.47, 41.07, 153.89) mm, rotated rx -180 ry 0 rz 180 deg; joints [-27.93, 59.725, -94.018, 32.688, 119.854, 17.715]
  MoveL 11245 to (237.47, 41.07, 153.89) mm, rotated rx -180 ry 0 rz 180 deg; joints [-27.93, 59.725, -94.018, 32.688, 119.854, 17.715]
  Call Extruder(205.52536)
  MoveL 11246 to (237.79, 41.51, 153.89) mm, rotated rx 180 ry 0 rz 180 deg; joints [-28.087, 59.784, -94.015, 32.842, 119.755, 17.763]
  MoveL 11247 to (237.79, 41.51, 153.89) mm, rotated rx 180 ry 0 rz 180 deg; joints [-28.087, 59.784, -94.015, 32.842, 119.755, 17.763]
  Call Extruder(205.85246)
  MoveL 11248 to (238.11, 41.96, 153.89) mm, rotated rx 180 ry 0 rz -180 deg; joints [-28.242, 59.843, -94.012, 32.992, 119.656, 17.808]
  MoveL 11249 to (238.11, 41.96, 153.89) mm, rotated rx 180 ry 0 rz -180 deg; joints [-28.242, 59.843, -94.012, 32.992, 119.656, 17.808]
  Call Extruder(205.98700)
  MoveL 11250 to (238.22, 42.15, 153.89) mm, rotated rx -180 ry 0 rz 180 deg; joints [-28.319, 59.866, -94.011, 33.069, 119.612, 17.834]
  MoveL 11251 to (238.22, 42.15, 153.89) mm, rotated rx -180 ry 0 rz 180 deg; joints [-28.319, 59.866, -94.011, 33.069, 119.612, 17.834]
  Call Extruder(206.20232)
  MoveL 11252 to (238.41, 42.47, 153.89) mm, rotated rx 180 ry 0 rz 180 deg; joints [-28.442, 59.903, -94.01, 33.192, 119.542, 17.877]
  MoveL 11253 to (238.41, 42.47, 153.89) mm, rotated rx 180 ry 0 rz 180 deg; joints [-28.442, 59.903, -94.01, 33.192, 119.542, 17.877]
  Call Extruder(206.41679)
  MoveL 11254 to (238.59, 42.79, 153.89) mm, rotated rx -180 ry 0 rz -180 deg; joints [-28.565, 59.939, -94.008, 33.314, 119.472, 17.919]
  MoveL 11255 to (238.59, 42.79, 153.89) mm, rotated rx -180 ry 0 rz -180 deg; joints [-28.565, 59.939, -94.008, 33.314, 119.472, 17.919]
  Call Extruder(206.63041)
  MoveL 11256 to (238.77, 43.1, 153.89) mm, rotated rx 180 ry 0 rz 180 deg; joints [-28.686, 59.976, -94.006, 33.435, 119.402, 17.96]
  MoveL 11257 to (238.77, 43.1, 153.89) mm, rotated rx 180 ry 0 rz 180 deg; joints [-28.686, 59.976, -94.006, 33.435, 119.402, 17.96]
  Call Extruder(206.80964)
  MoveL 11258 to (238.91, 43.37, 153.89) mm, rotated rx 180 ry 0 rz 180 deg; joints [-28.796, 60.006, -94.005, 33.544, 119.342, 17.998]
  MoveL 11259 to (238.91, 43.37, 153.89) mm, rotated rx 180 ry 0 rz 180 deg; joints [-28.796, 60.006, -94.005, 33.544, 119.342, 17.998]
  Call Extruder(206.95538)
  MoveL 11260 to (239.01, 43.6, 153.89) mm, rotated rx 180 ry 0 rz -180 deg; joints [-28.894, 60.03, -94.003, 33.644, 119.291, 18.035]
  MoveL 11261 to (239.01, 43.6, 153.89) mm, rotated rx 180 ry 0 rz -180 deg; joints [-28.894, 60.03, -94.003, 33.644, 119.291, 18.035]
  Call Extruder(207.10061)
  MoveL 11262 to (239.11, 43.83, 153.89) mm, rotated rx 180 ry 0 rz 180 deg; joints [-28.991, 60.053, -94.002, 33.742, 119.24, 18.071]
  MoveL 11263 to (239.11, 43.83, 153.89) mm, rotated rx 180 ry 0 rz 180 deg; joints [-28.991, 60.053, -94.002, 33.742, 119.24, 18.071]
  Call Extruder(207.28332)
  MoveL 11264 to (239.22, 44.12, 153.89) mm, rotated rx -180 ry 0 rz 180 deg; joints [-29.116, 60.083, -94.001, 33.868, 119.176, 18.118]
  MoveL 11265 to (239.22, 44.12, 153.89) mm, rotated rx -180 ry 0 rz 180 deg; joints [-29.116, 60.083, -94.001, 33.868, 119.176, 18.118]
  Call Extruder(207.46527)
  MoveL 11266 to (239.35, 44.42, 153.89) mm, rotated rx 180 ry 0 rz 180 deg; joints [-29.24, 60.112, -93.999, 33.993, 119.112, 18.163]
  MoveL 11267 to (239.35, 44.42, 153.89) mm, rotated rx 180 ry 0 rz 180 deg; joints [-29.24, 60.112, -93.999, 33.993, 119.112, 18.163]
  Call Extruder(207.61260)
  MoveL 11268 to (239.44, 44.66, 153.89) mm, rotated rx 180 ry 0 rz 180 deg; joints [-29.343, 60.135, -93.998, 34.098, 119.059, 18.202]
  MoveL 11269 to (239.44, 44.66, 153.89) mm, rotated rx 180 ry 0 rz 180 deg; joints [-29.343, 60.135, -93.998, 34.098, 119.059, 18.202]
  Call Extruder(207.72584)
  MoveL 11270 to (239.5, 44.85, 153.89) mm, rotated rx 180 ry 0 rz 180 deg; joints [-29.428, 60.153, -93.997, 34.184, 119.018, 18.235]
  MoveL 11271 to (239.5, 44.85, 153.89) mm, rotated rx 180 ry 0 rz 180 deg; joints [-29.428, 60.153, -93.997, 34.184, 119.018, 18.235]
  Call Extruder(207.83863)
  MoveL 11272 to (239.56, 45.03, 153.89) mm, rotated rx 180 ry 0 rz 180 deg; joints [-29.512, 60.17, -93.996, 34.269, 118.976, 18.268]
  MoveL 11273 to (239.56, 45.03, 153.89) mm, rotated rx 180 ry 0 rz 180 deg; joints [-29.512, 60.17, -93.996, 34.269, 118.976, 18.268]
  Call Extruder(207.95098)
  MoveL 11274 to (239.62, 45.22, 153.89) mm, rotated rx -180 ry 0 rz -180 deg; joints [-29.596, 60.187, -93.995, 34.355, 118.935, 18.3]
  MoveL 11275 to (239.62, 45.22, 153.89) mm, rotated rx -180 ry 0 rz -180 deg; joints [-29.596, 60.187, -93.995, 34.355, 118.935, 18.3]
  Call Extruder(208.06288)
  MoveL 11276 to (239.68, 45.41, 153.89) mm, rotated rx -180 ry 0 rz 180 deg; joints [-29.679, 60.205, -93.994, 34.44, 118.894, 18.332]
  MoveL 11277 to (239.68, 45.41, 153.89) mm, rotated rx -180 ry 0 rz 180 deg; joints [-29.679, 60.205, -93.994, 34.44, 118.894, 18.332]
  Call Extruder(208.18428)
  MoveL 11278 to (239.75, 45.62, 153.89) mm, rotated rx -180 ry 0 rz 180 deg; joints [-29.77, 60.223, -93.993, 34.533, 118.848, 18.367]
  MoveL 11279 to (239.75, 45.62, 153.89) mm, rotated rx -180 ry 0 rz 180 deg; joints [-29.77, 60.223, -93.993, 34.533, 118.848, 18.367]
  Call Extruder(208.31507)
  MoveL 11280 to (239.82, 45.84, 153.89) mm, rotated rx -180 ry 0 rz 180 deg; joints [-29.871, 60.244, -93.992, 34.634, 118.799, 18.405]
  MoveL 11281 to (239.82, 45.84, 153.89) mm, rotated rx -180 ry 0 rz 180 deg; joints [-29.871, 60.244, -93.992, 34.634, 118.799, 18.405]
  Call Extruder(208.44530)
  MoveL 11282 to (239.88, 46.06, 153.89) mm, rotated rx -180 ry 0 rz -180 deg; joints [-29.97, 60.264, -93.991, 34.735, 118.75, 18.443]
  MoveL 11283 to (239.88, 46.06, 153.89) mm, rotated rx -180 ry 0 rz -180 deg; joints [-29.97, 60.264, -93.991, 34.735, 118.75, 18.443]
  Call Extruder(208.57496)
  MoveL 11284 to (239.95, 46.29, 153.89) mm, rotated rx -180 ry 0 rz 180 deg; joints [-30.069, 60.284, -93.99, 34.836, 118.701, 18.481]
  MoveL 11285 to (239.95, 46.29, 153.89) mm, rotated rx -180 ry 0 rz 180 deg; joints [-30.069, 60.284, -93.99, 34.836, 118.701, 18.481]
  Call Extruder(208.70405)
  MoveL 11286 to (240.02, 46.51, 153.89) mm, rotated rx 180 ry 0 rz 180 deg; joints [-30.168, 60.304, -93.988, 34.937, 118.653, 18.519]
  MoveL 11287 to (240.02, 46.51, 153.89) mm, rotated rx 180 ry 0 rz 180 deg; joints [-30.168, 60.304, -93.988, 34.937, 118.653, 18.519]
  Call Extruder(208.81911)
  MoveL 11288 to (240.06, 46.72, 153.89) mm, rotated rx -180 ry 0 rz 180 deg; joints [-30.263, 60.321, -93.987, 35.034, 118.608, 18.556]
  MoveL 11289 to (240.06, 46.72, 153.89) mm, rotated rx -180 ry 0 rz 180 deg; joints [-30.263, 60.321, -93.987, 35.034, 118.608, 18.556]
  Call Extruder(208.93371)
  MoveL 11290 to (240.11, 46.92, 153.89) mm, rotated rx -180 ry 0 rz 180 deg; joints [-30.358, 60.337, -93.986, 35.131, 118.563, 18.594]
  MoveL 11291 to (240.11, 46.92, 153.89) mm, rotated rx -180 ry 0 rz 180 deg; joints [-30.358, 60.337, -93.986, 35.131, 118.563, 18.594]
  Call Extruder(209.04786)
  MoveL 11292 to (240.15, 47.12, 153.89) mm, rotated rx -180 ry 0 rz 180 deg; joints [-30.453, 60.354, -93.985, 35.227, 118.518, 18.631]
  MoveL 11293 to (240.15, 47.12, 153.89) mm, rotated rx -180 ry 0 rz 180 deg; joints [-30.453, 60.354, -93.985, 35.227, 118.518, 18.631]
  Call Extruder(209.16155)
  MoveL 11294 to (240.2, 47.33, 153.89) mm, rotated rx -180 ry 0 rz 180 deg; joints [-30.548, 60.371, -93.984, 35.324, 118.474, 18.668]
  MoveL 11295 to (240.2, 47.33, 153.89) mm, rotated rx -180 ry 0 rz 180 deg; joints [-30.548, 60.371, -93.984, 35.324, 118.474, 18.668]
  Call Extruder(209.28696)
  MoveL 11296 to (240.24, 47.56, 153.89) mm, rotated rx -180 ry 0 rz 180 deg; joints [-30.653, 60.389, -93.983, 35.431, 118.424, 18.709]
  MoveL 11297 to (240.24, 47.56, 153.89) mm, rotated rx -180 ry 0 rz 180 deg; joints [-30.653, 60.389, -93.983, 35.431, 118.424, 18.709]
  Call Extruder(209.42394)
  MoveL 11298 to (240.29, 47.8, 153.89) mm, rotated rx 180 ry 0 rz 180 deg; joints [-30.768, 60.409, -93.982, 35.548, 118.37, 18.754]
  MoveL 11299 to (240.29, 47.8, 153.89) mm, rotated rx 180 ry 0 rz 180 deg; joints [-30.768, 60.409, -93.982, 35.548, 118.37, 18.754]
  Call Extruder(209.56031)
  MoveL 11300 to (240.34, 48.05, 153.89) mm, rotated rx 180 ry 0 rz 180 deg; joints [-30.884, 60.429, -93.981, 35.666, 118.315, 18.799]
  MoveL 11301 to (240.34, 48.05, 153.89) mm, rotated rx 180 ry 0 rz 180 deg; joints [-30.884, 60.429, -93.981, 35.666, 118.315, 18.799]
  Call Extruder(209.69607)
  MoveL 11302 to (240.39, 48.3, 153.89) mm, rotated rx 180 ry 0 rz 180 deg; joints [-30.999, 60.45, -93.98, 35.783, 118.26, 18.844]
  MoveL 11303 to (240.39, 48.3, 153.89) mm, rotated rx 180 ry 0 rz 180 deg; joints [-30.999, 60.45, -93.98, 35.783, 118.26, 18.844]
  Call Extruder(209.83121)
  MoveL 11304 to (240.44, 48.55, 153.89) mm, rotated rx 180 ry 0 rz 180 deg; joints [-31.114, 60.47, -93.978, 35.9, 118.206, 18.888]
  MoveL 11305 to (240.44, 48.55, 153.89) mm, rotated rx 180 ry 0 rz 180 deg; joints [-31.114, 60.47, -93.978, 35.9, 118.206, 18.888]
  Call Extruder(209.96575)
  MoveL 11306 to (240.49, 48.8, 153.89) mm, rotated rx 180 ry 0 rz 180 deg; joints [-31.228, 60.49, -93.977, 36.016, 118.152, 18.931]
  MoveL 11307 to (240.49, 48.8, 153.89) mm, rotated rx 180 ry 0 rz 180 deg; joints [-31.228, 60.49, -93.977, 36.016, 118.152, 18.931]
  Call Extruder(210.09968)
  MoveL 11308 to (240.54, 49.05, 153.89) mm, rotated rx 180 ry 0 rz 180 deg; joints [-31.342, 60.51, -93.976, 36.131, 118.097, 18.974]
  MoveL 11309 to (240.54, 49.05, 153.89) mm, rotated rx 180 ry 0 rz 180 deg; joints [-31.342, 60.51, -93.976, 36.131, 118.097, 18.974]
  Call Extruder(210.24754)
  MoveL 11310 to (240.59, 49.33, 153.89) mm, rotated rx 180 ry 0 rz 180 deg; joints [-31.47, 60.532, -93.974, 36.261, 118.037, 19.023]
  MoveL 11311 to (240.59, 49.33, 153.89) mm, rotated rx 180 ry 0 rz 180 deg; joints [-31.47, 60.532, -93.974, 36.261, 118.037, 19.023]
  Call Extruder(210.40929)
  MoveL 11312 to (240.64, 49.63, 153.89) mm, rotated rx 180 ry 0 rz 180 deg; joints [-31.612, 60.556, -93.973, 36.405, 117.97, 19.078]
  MoveL 11313 to (240.64, 49.63, 153.89) mm, rotated rx 180 ry 0 rz 180 deg; joints [-31.612, 60.556, -93.973, 36.405, 117.97, 19.078]
  Call Extruder(210.57031)
  MoveL 11314 to (240.69, 49.94, 153.89) mm, rotated rx 180 ry 0 rz 180 deg; joints [-31.755, 60.58, -93.971, 36.549, 117.903, 19.132]
  MoveL 11315 to (240.69, 49.94, 153.89) mm, rotated rx 180 ry 0 rz 180 deg; joints [-31.755, 60.58, -93.971, 36.549, 117.903, 19.132]
  Call Extruder(210.73060)
  MoveL 11316 to (240.74, 50.24, 153.89) mm, rotated rx 180 ry 0 rz 180 deg; joints [-31.895, 60.603, -93.97, 36.692, 117.836, 19.185]
  MoveL 11317 to (240.74, 50.24, 153.89) mm, rotated rx 180 ry 0 rz 180 deg; joints [-31.895, 60.603, -93.97, 36.692, 117.836, 19.185]
  Call Extruder(210.89016)
  MoveL 11318 to (240.78, 50.55, 153.89) mm, rotated rx 180 ry 0 rz 180 deg; joints [-32.036, 60.627, -93.968, 36.834, 117.77, 19.238]
  MoveL 11319 to (240.78, 50.55, 153.89) mm, rotated rx 180 ry 0 rz 180 deg; joints [-32.036, 60.627, -93.968, 36.834, 117.77, 19.238]
  Call Extruder(211.04899)
  MoveL 11320 to (240.83, 50.86, 153.89) mm, rotated rx 180 ry 0 rz 180 deg; joints [-32.176, 60.651, -93.966, 36.976, 117.703, 19.29]
  MoveL 11321 to (240.83, 50.86, 153.89) mm, rotated rx 180 ry 0 rz 180 deg; joints [-32.176, 60.651, -93.966, 36.976, 117.703, 19.29]
  Call Extruder(211.22766)
  MoveL 11322 to (240.88, 51.2, 153.89) mm, rotated rx 180 ry 0 rz 180 deg; joints [-32.337, 60.678, -93.965, 37.137, 117.627, 19.351]
  MoveL 11323 to (240.88, 51.2, 153.89) mm, rotated rx 180 ry 0 rz 180 deg; joints [-32.337, 60.678, -93.965, 37.137, 117.627, 19.351]
  Call Extruder(211.42611)
  MoveL 11324 to (240.93, 51.59, 153.89) mm, rotated rx 180 ry 0 rz 180 deg; joints [-32.518, 60.706, -93.962, 37.32, 117.543, 19.419]
  MoveL 11325 to (240.93, 51.59, 153.89) mm, rotated rx 180 ry 0 rz 180 deg; joints [-32.518, 60.706, -93.962, 37.32, 117.543, 19.419]
  Call Extruder(211.62368)
  MoveL 11326 to (240.97, 51.98, 153.89) mm, rotated rx 180 ry 0 rz 180 deg; joints [-32.697, 60.735, -93.96, 37.501, 117.458, 19.485]
  MoveL 11327 to (240.97, 51.98, 153.89) mm, rotated rx 180 ry 0 rz 180 deg; joints [-32.697, 60.735, -93.96, 37.501, 117.458, 19.485]
  Call Extruder(211.82039)
  MoveL 11328 to (241.02, 52.37, 153.89) mm, rotated rx 180 ry 0 rz 180 deg; joints [-32.876, 60.765, -93.958, 37.682, 117.374, 19.552]
  MoveL 11329 to (241.02, 52.37, 153.89) mm, rotated rx 180 ry 0 rz 180 deg; joints [-32.876, 60.765, -93.958, 37.682, 117.374, 19.552]
  Call Extruder(212.01622)
  MoveL 11330 to (241.06, 52.75, 153.89) mm, rotated rx -180 ry 0 rz 180 deg; joints [-33.055, 60.794, -93.956, 37.861, 117.289, 19.617]
  MoveL 11331 to (241.06, 52.75, 153.89) mm, rotated rx -180 ry 0 rz 180 deg; joints [-33.055, 60.794, -93.956, 37.861, 117.289, 19.617]
  Call Extruder(212.31166)
  MoveL 11332 to (241.11, 53.34, 153.89) mm, rotated rx -180 ry 0 rz 180 deg; joints [-33.331, 60.836, -93.953, 38.139, 117.16, 19.719]
  MoveL 11333 to (241.11, 53.34, 153.89) mm, rotated rx -180 ry 0 rz 180 deg; joints [-33.331, 60.836, -93.953, 38.139, 117.16, 19.719]
  Call Extruder(212.60577)
  MoveL 11334 to (241.16, 53.93, 153.89) mm, rotated rx 180 ry 0 rz 180 deg; joints [-33.606, 60.879, -93.95, 38.415, 117.031, 19.82]
  MoveL 11335 to (241.16, 53.93, 153.89) mm, rotated rx 180 ry 0 rz 180 deg; joints [-33.606, 60.879, -93.95, 38.415, 117.031, 19.82]
  Call Extruder(212.89854)
  MoveL 11336 to (241.2, 54.52, 153.89) mm, rotated rx 180 ry 0 rz 180 deg; joints [-33.878, 60.922, -93.947, 38.688, 116.903, 19.918]
  MoveL 11337 to (241.2, 54.52, 153.89) mm, rotated rx 180 ry 0 rz 180 deg; joints [-33.878, 60.922, -93.947, 38.688, 116.903, 19.918]
  Call Extruder(213.47199)
  MoveL 11338 to (241.25, 55.68, 153.89) mm, rotated rx 180 ry 0 rz 180 deg; joints [-34.425, 61.002, -93.94, 39.235, 116.648, 20.116]
  MoveL 11339 to (241.25, 55.68, 153.89) mm, rotated rx 180 ry 0 rz 180 deg; joints [-34.425, 61.002, -93.94, 39.235, 116.648, 20.116]
  Call Extruder(214.18582)
  MoveL 11340 to (241.29, 57.14, 153.89) mm, rotated rx -180 ry 0 rz 180 deg; joints [-35.104, 61.103, -93.932, 39.913, 116.329, 20.356]
  Call Extruder(256.25069)
  MoveL 11341 to (241.29, 142.86, 153.89) mm, rotated rx 180 ry 0 rz 180 deg; joints [-60.361, 68.082, -92.479, 62.608, 101.787, 21.515]
  Call Extruder(256.67912)
  MoveL 11342 to (241.27, 143.73, 153.89) mm, rotated rx 180 ry 0 rz 180 deg; joints [-60.516, 68.156, -92.453, 62.736, 101.684, 21.454]
  MoveL 11343 to (241.27, 143.73, 153.89) mm, rotated rx 180 ry 0 rz 180 deg; joints [-60.516, 68.156, -92.453, 62.736, 101.684, 21.454]
  Call Extruder(257.25257)
  MoveL 11344 to (241.23, 144.9, 153.89) mm, rotated rx 180 ry 0 rz 180 deg; joints [-60.726, 68.252, -92.417, 62.913, 101.547, 21.375]
  MoveL 11345 to (241.23, 144.9, 153.89) mm, rotated rx 180 ry 0 rz 180 deg; joints [-60.726, 68.252, -92.417, 62.913, 101.547, 21.375]
  Call Extruder(257.68690)
  MoveL 11346 to (241.18, 145.77, 153.89) mm, rotated rx -180 ry 0 rz 180 deg; joints [-60.887, 68.324, -92.391, 63.048, 101.444, 21.316]
  MoveL 11347 to (241.18, 145.77, 153.89) mm, rotated rx -180 ry 0 rz 180 deg; joints [-60.887, 68.324, -92.391, 63.048, 101.444, 21.316]
  Call Extruder(257.98101)
  MoveL 11348 to (241.13, 146.36, 153.89) mm, rotated rx -180 ry 0 rz 180 deg; joints [-61, 68.372, -92.373, 63.143, 101.374, 21.277]
  MoveL 11349 to (241.13, 146.36, 153.89) mm, rotated rx -180 ry 0 rz 180 deg; joints [-61, 68.372, -92.373, 63.143, 101.374, 21.277]
  Call Extruder(258.27645)
  MoveL 11350 to (241.09, 146.95, 153.89) mm, rotated rx 180 ry 0 rz 180 deg; joints [-61.111, 68.419, -92.355, 63.237, 101.304, 21.239]
  MoveL 11351 to (241.09, 146.95, 153.89) mm, rotated rx 180 ry 0 rz 180 deg; joints [-61.111, 68.419, -92.355, 63.237, 101.304, 21.239]
  Call Extruder(258.52270)
  MoveL 11352 to (241.04, 147.44, 153.89) mm, rotated rx -180 ry 0 rz -180 deg; joints [-61.205, 68.458, -92.34, 63.317, 101.245, 21.207]
  MoveL 11353 to (241.04, 147.44, 153.89) mm, rotated rx -180 ry 0 rz -180 deg; joints [-61.205, 68.458, -92.34, 63.317, 101.245, 21.207]
  Call Extruder(258.71941)
  MoveL 11354 to (240.99, 147.83, 153.89) mm, rotated rx 180 ry 0 rz 180 deg; joints [-61.282, 68.489, -92.329, 63.383, 101.198, 21.183]
  MoveL 11355 to (240.99, 147.83, 153.89) mm, rotated rx 180 ry 0 rz 180 deg; joints [-61.282, 68.489, -92.329, 63.383, 101.198, 21.183]
  Call Extruder(258.91698)
  MoveL 11356 to (240.95, 148.22, 153.89) mm, rotated rx 180 ry 0 rz 180 deg; joints [-61.359, 68.52, -92.317, 63.448, 101.152, 21.158]
  MoveL 11357 to (240.95, 148.22, 153.89) mm, rotated rx 180 ry 0 rz 180 deg; joints [-61.359, 68.52, -92.317, 63.448, 101.152, 21.158]
  Call Extruder(259.11542)
  MoveL 11358 to (240.9, 148.6, 153.89) mm, rotated rx 180 ry 0 rz 180 deg; joints [-61.436, 68.55, -92.305, 63.513, 101.105, 21.134]
  MoveL 11359 to (240.9, 148.6, 153.89) mm, rotated rx 180 ry 0 rz 180 deg; joints [-61.436, 68.55, -92.305, 63.513, 101.105, 21.134]
  Call Extruder(259.31473)
  MoveL 11360 to (240.86, 148.99, 153.89) mm, rotated rx 180 ry 0 rz 180 deg; joints [-61.512, 68.581, -92.294, 63.578, 101.059, 21.109]
  MoveL 11361 to (240.86, 148.99, 153.89) mm, rotated rx 180 ry 0 rz 180 deg; joints [-61.512, 68.581, -92.294, 63.578, 101.059, 21.109]
  Call Extruder(259.47356)
  MoveL 11362 to (240.81, 149.3, 153.89) mm, rotated rx 180 ry 0 rz 180 deg; joints [-61.575, 68.604, -92.285, 63.633, 101.022, 21.091]
  MoveL 11363 to (240.81, 149.3, 153.89) mm, rotated rx 180 ry 0 rz 180 deg; joints [-61.575, 68.604, -92.285, 63.633, 101.022, 21.091]
  Call Extruder(259.63312)
  MoveL 11364 to (240.76, 149.6, 153.89) mm, rotated rx 180 ry 0 rz 180 deg; joints [-61.639, 68.628, -92.275, 63.688, 100.984, 21.073]
  MoveL 11365 to (240.76, 149.6, 153.89) mm, rotated rx 180 ry 0 rz 180 deg; joints [-61.639, 68.628, -92.275, 63.688, 100.984, 21.073]
  Call Extruder(259.79341)
  MoveL 11366 to (240.71, 149.91, 153.89) mm, rotated rx 180 ry 0 rz -180 deg; joints [-61.702, 68.652, -92.266, 63.742, 100.947, 21.054]
  MoveL 11367 to (240.71, 149.91, 153.89) mm, rotated rx 180 ry 0 rz -180 deg; joints [-61.702, 68.652, -92.266, 63.742, 100.947, 21.054]
  Call Extruder(259.95443)
  MoveL 11368 to (240.66, 150.21, 153.89) mm, rotated rx 180 ry 0 rz 180 deg; joints [-61.765, 68.675, -92.257, 63.797, 100.91, 21.036]
  MoveL 11369 to (240.66, 150.21, 153.89) mm, rotated rx 180 ry 0 rz 180 deg; joints [-61.765, 68.675, -92.257, 63.797, 100.91, 21.036]
  Call Extruder(260.11618)
  MoveL 11370 to (240.61, 150.52, 153.89) mm, rotated rx -180 ry 0 rz 180 deg; joints [-61.828, 68.699, -92.248, 63.851, 100.873, 21.017]
  MoveL 11371 to (240.61, 150.52, 153.89) mm, rotated rx -180 ry 0 rz 180 deg; joints [-61.828, 68.699, -92.248, 63.851, 100.873, 21.017]
  Call Extruder(260.27865)
  MoveL 11372 to (240.56, 150.83, 153.89) mm, rotated rx -180 ry 0 rz 180 deg; joints [-61.891, 68.722, -92.239, 63.905, 100.836, 20.998]
  MoveL 11373 to (240.56, 150.83, 153.89) mm, rotated rx -180 ry 0 rz 180 deg; joints [-61.891, 68.722, -92.239, 63.905, 100.836, 20.998]
  Call Extruder(260.41257)
  MoveL 11374 to (240.52, 151.07, 153.89) mm, rotated rx -180 ry 0 rz 180 deg; joints [-61.944, 68.741, -92.231, 63.951, 100.805, 20.984]
  MoveL 11375 to (240.52, 151.07, 153.89) mm, rotated rx -180 ry 0 rz 180 deg; joints [-61.944, 68.741, -92.231, 63.951, 100.805, 20.984]
  Call Extruder(260.54711)
  MoveL 11376 to (240.47, 151.32, 153.89) mm, rotated rx 180 ry 0 rz 180 deg; joints [-61.998, 68.76, -92.224, 63.998, 100.774, 20.969]
  MoveL 11377 to (240.47, 151.32, 153.89) mm, rotated rx 180 ry 0 rz 180 deg; joints [-61.998, 68.76, -92.224, 63.998, 100.774, 20.969]
  Call Extruder(260.68226)
  MoveL 11378 to (240.42, 151.57, 153.89) mm, rotated rx 180 ry 0 rz 180 deg; joints [-62.052, 68.779, -92.216, 64.045, 100.744, 20.955]
  MoveL 11379 to (240.42, 151.57, 153.89) mm, rotated rx 180 ry 0 rz 180 deg; joints [-62.052, 68.779, -92.216, 64.045, 100.744, 20.955]
  Call Extruder(260.81801)
  MoveL 11380 to (240.37, 151.82, 153.89) mm, rotated rx 180 ry 0 rz -180 deg; joints [-62.105, 68.797, -92.209, 64.091, 100.713, 20.94]
  MoveL 11381 to (240.37, 151.82, 153.89) mm, rotated rx 180 ry 0 rz -180 deg; joints [-62.105, 68.797, -92.209, 64.091, 100.713, 20.94]
  Call Extruder(260.95438)
  MoveL 11382 to (240.32, 152.07, 153.89) mm, rotated rx 180 ry 0 rz 180 deg; joints [-62.159, 68.816, -92.201, 64.137, 100.682, 20.926]
  MoveL 11383 to (240.32, 152.07, 153.89) mm, rotated rx 180 ry 0 rz 180 deg; joints [-62.159, 68.816, -92.201, 64.137, 100.682, 20.926]
  Call Extruder(261.09136)
  MoveL 11384 to (240.27, 152.32, 153.89) mm, rotated rx -180 ry 0 rz 180 deg; joints [-62.212, 68.835, -92.194, 64.183, 100.652, 20.911]
  MoveL 11385 to (240.27, 152.32, 153.89) mm, rotated rx -180 ry 0 rz 180 deg; joints [-62.212, 68.835, -92.194, 64.183, 100.652, 20.911]
  Call Extruder(261.22895)
  MoveL 11386 to (240.22, 152.57, 153.89) mm, rotated rx 180 ry 0 rz 180 deg; joints [-62.265, 68.854, -92.186, 64.23, 100.622, 20.896]
  MoveL 11387 to (240.22, 152.57, 153.89) mm, rotated rx 180 ry 0 rz 180 deg; joints [-62.265, 68.854, -92.186, 64.23, 100.622, 20.896]
  Call Extruder(261.34265)
  MoveL 11388 to (240.17, 152.77, 153.89) mm, rotated rx 180 ry 0 rz 180 deg; joints [-62.31, 68.869, -92.18, 64.268, 100.596, 20.885]
  MoveL 11389 to (240.17, 152.77, 153.89) mm, rotated rx 180 ry 0 rz 180 deg; joints [-62.31, 68.869, -92.18, 64.268, 100.596, 20.885]
  Call Extruder(261.45680)
  MoveL 11390 to (240.13, 152.98, 153.89) mm, rotated rx 180 ry 0 rz -180 deg; joints [-62.355, 68.884, -92.174, 64.307, 100.571, 20.873]
  MoveL 11391 to (240.13, 152.98, 153.89) mm, rotated rx 180 ry 0 rz -180 deg; joints [-62.355, 68.884, -92.174, 64.307, 100.571, 20.873]
  Call Extruder(261.57140)
  MoveL 11392 to (240.08, 153.18, 153.89) mm, rotated rx 180 ry 0 rz 180 deg; joints [-62.399, 68.899, -92.168, 64.346, 100.546, 20.861]
  MoveL 11393 to (240.08, 153.18, 153.89) mm, rotated rx 180 ry 0 rz 180 deg; joints [-62.399, 68.899, -92.168, 64.346, 100.546, 20.861]
  Call Extruder(261.68645)
  MoveL 11394 to (240.04, 153.39, 153.89) mm, rotated rx -180 ry 0 rz -180 deg; joints [-62.444, 68.914, -92.162, 64.384, 100.521, 20.849]
  MoveL 11395 to (240.04, 153.39, 153.89) mm, rotated rx -180 ry 0 rz -180 deg; joints [-62.444, 68.914, -92.162, 64.384, 100.521, 20.849]
  Call Extruder(261.80867)
  MoveL 11396 to (239.98, 153.6, 153.89) mm, rotated rx 180 ry 0 rz 180 deg; joints [-62.493, 68.93, -92.156, 64.428, 100.494, 20.838]
  MoveL 11397 to (239.98, 153.6, 153.89) mm, rotated rx 180 ry 0 rz 180 deg; joints [-62.493, 68.93, -92.156, 64.428, 100.494, 20.838]
  Call Extruder(261.93833)
  MoveL 11398 to (239.92, 153.82, 153.89) mm, rotated rx 180 ry 0 rz 180 deg; joints [-62.547, 68.946, -92.149, 64.475, 100.465, 20.827]
  MoveL 11399 to (239.92, 153.82, 153.89) mm, rotated rx 180 ry 0 rz 180 deg; joints [-62.547, 68.946, -92.149, 64.475, 100.465, 20.827]
  Call Extruder(262.06856)
  MoveL 11400 to (239.85, 154.05, 153.89) mm, rotated rx -180 ry 0 rz 180 deg; joints [-62.601, 68.962, -92.143, 64.523, 100.437, 20.816]
  MoveL 11401 to (239.85, 154.05, 153.89) mm, rotated rx -180 ry 0 rz 180 deg; joints [-62.601, 68.962, -92.143, 64.523, 100.437, 20.816]
  Call Extruder(262.19935)
  MoveL 11402 to (239.78, 154.27, 153.89) mm, rotated rx 180 ry 0 rz 180 deg; joints [-62.654, 68.978, -92.136, 64.57, 100.408, 20.804]
  MoveL 11403 to (239.78, 154.27, 153.89) mm, rotated rx 180 ry 0 rz 180 deg; joints [-62.654, 68.978, -92.136, 64.57, 100.408, 20.804]
  Call Extruder(262.33071)
  MoveL 11404 to (239.71, 154.5, 153.89) mm, rotated rx 180 ry 0 rz 180 deg; joints [-62.708, 68.993, -92.13, 64.617, 100.379, 20.793]
  MoveL 11405 to (239.71, 154.5, 153.89) mm, rotated rx 180 ry 0 rz 180 deg; joints [-62.708, 68.993, -92.13, 64.617, 100.379, 20.793]
  Call Extruder(262.44261)
  MoveL 11406 to (239.65, 154.68, 153.89) mm, rotated rx 180 ry 0 rz 180 deg; joints [-62.754, 69.007, -92.124, 64.658, 100.355, 20.784]
  MoveL 11407 to (239.65, 154.68, 153.89) mm, rotated rx 180 ry 0 rz 180 deg; joints [-62.754, 69.007, -92.124, 64.658, 100.355, 20.784]
  Call Extruder(262.55495)
  MoveL 11408 to (239.59, 154.87, 153.89) mm, rotated rx -180 ry 0 rz -180 deg; joints [-62.801, 69.02, -92.119, 64.699, 100.331, 20.775]
  MoveL 11409 to (239.59, 154.87, 153.89) mm, rotated rx -180 ry 0 rz -180 deg; joints [-62.801, 69.02, -92.119, 64.699, 100.331, 20.775]
  Call Extruder(262.66774)
  MoveL 11410 to (239.53, 155.06, 153.89) mm, rotated rx 180 ry 0 rz -180 deg; joints [-62.847, 69.033, -92.114, 64.74, 100.306, 20.765]
  MoveL 11411 to (239.53, 155.06, 153.89) mm, rotated rx 180 ry 0 rz -180 deg; joints [-62.847, 69.033, -92.114, 64.74, 100.306, 20.765]
  Call Extruder(262.78098)
